REGION Network 2: Manual Operation Cm - typeAxis64PosInterface
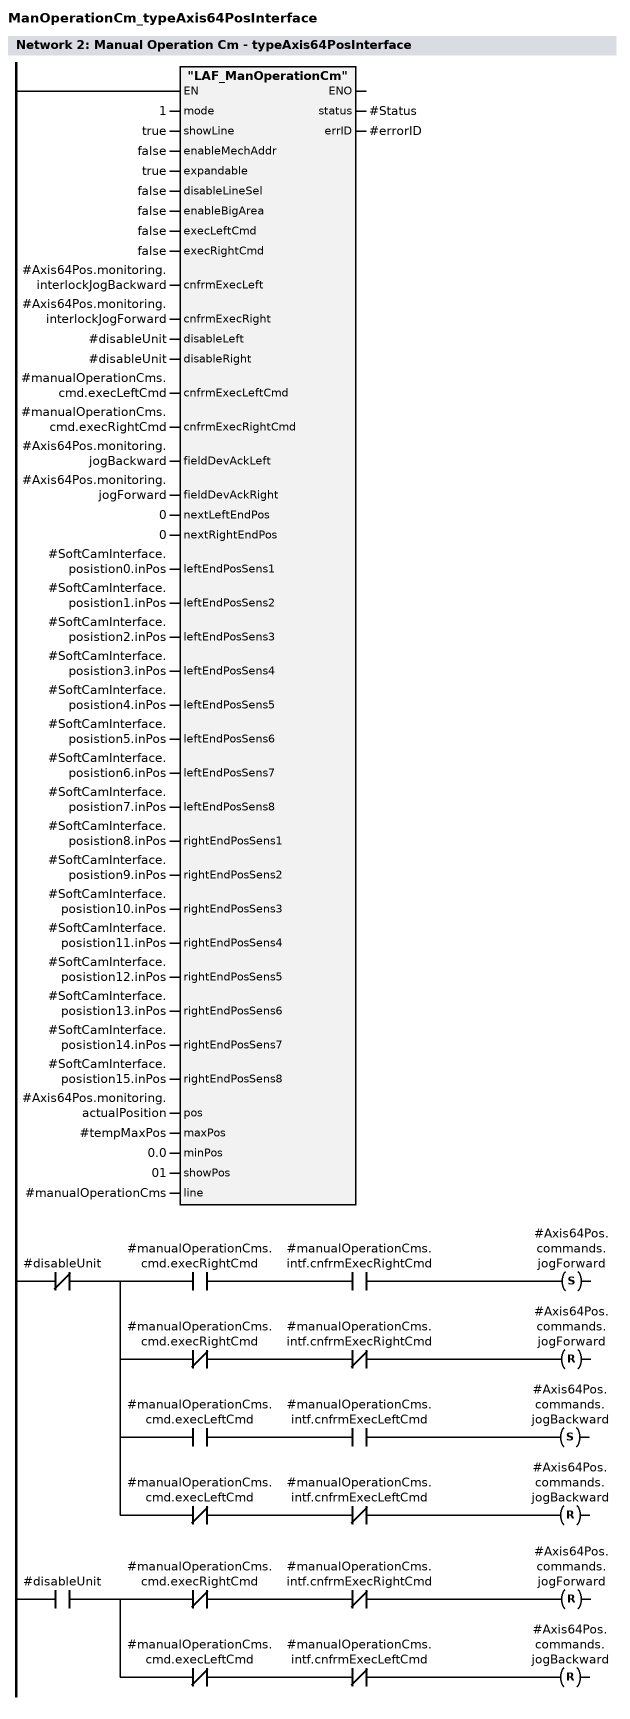
   RUNG wire#powerrail
      "LAF_ManOperationCm"(mode := 1, showLine := true, enableMechAddr := false, expandable := true, disableLineSel := false, enableBigArea := false, execLeftCmd := false, execRightCmd := false, cnfrmExecLeft := #Axis64Pos.monitoring.interlockJogBackward, cnfrmExecRight := #Axis64Pos.monitoring.interlockJogForward, disableLeft := #disableUnit, disableRight := #disableUnit, cnfrmExecLeftCmd := #manualOperationCms.cmd.execLeftCmd, cnfrmExecRightCmd := #manualOperationCms.cmd.execRightCmd, fieldDevAckLeft := #Axis64Pos.monitoring.jogBackward, fieldDevAckRight := #Axis64Pos.monitoring.jogForward, nextLeftEndPos := 0, nextRightEndPos := 0, leftEndPosSens1 := #SoftCamInterface.posistion0.inPos, leftEndPosSens2 := #SoftCamInterface.posistion1.inPos, leftEndPosSens3 := #SoftCamInterface.posistion2.inPos, leftEndPosSens4 := #SoftCamInterface.posistion3.inPos, leftEndPosSens5 := #SoftCamInterface.posistion4.inPos, leftEndPosSens6 := #SoftCamInterface.posistion5.inPos, leftEndPosSens7 := #SoftCamInterface.posistion6.inPos, leftEndPosSens8 := #SoftCamInterface.posistion7.inPos, rightEndPosSens1 := #SoftCamInterface.posistion8.inPos, rightEndPosSens2 := #SoftCamInterface.posistion9.inPos, rightEndPosSens3 := #SoftCamInterface.posistion10.inPos, rightEndPosSens4 := #SoftCamInterface.posistion11.inPos, rightEndPosSens5 := #SoftCamInterface.posistion12.inPos, rightEndPosSens6 := #SoftCamInterface.posistion13.inPos, rightEndPosSens7 := #SoftCamInterface.posistion14.inPos, rightEndPosSens8 := #SoftCamInterface.posistion15.inPos, pos := #Axis64Pos.monitoring.actualPosition, maxPos := #tempMaxPos, minPos := 0.0, showPos := 01, line := #manualOperationCms, status => #Status, errID => #errorID)
   END_RUNG
   RUNG wire#powerrail
      I_Contact( #disableUnit )
      wire#w1
      Contact( #manualOperationCms.cmd.execRightCmd )
      Contact( #manualOperationCms.intf.cnfrmExecRightCmd )
      S_Coil( #Axis64Pos.commands.jogForward )
   END_RUNG
   RUNG wire#w1
      I_Contact( #manualOperationCms.cmd.execRightCmd )
      I_Contact( #manualOperationCms.intf.cnfrmExecRightCmd )
      R_Coil( #Axis64Pos.commands.jogForward )
   END_RUNG
   RUNG wire#w1
      Contact( #manualOperationCms.cmd.execLeftCmd )
      Contact( #manualOperationCms.intf.cnfrmExecLeftCmd )
      S_Coil( #Axis64Pos.commands.jogBackward )
   END_RUNG
   RUNG wire#w1
      I_Contact( #manualOperationCms.cmd.execLeftCmd )
      I_Contact( #manualOperationCms.intf.cnfrmExecLeftCmd )
      R_Coil( #Axis64Pos.commands.jogBackward )
   END_RUNG
   RUNG wire#powerrail
      Contact( #disableUnit )
      wire#w2
      I_Contact( #manualOperationCms.cmd.execRightCmd )
      I_Contact( #manualOperationCms.intf.cnfrmExecRightCmd )
      R_Coil( #Axis64Pos.commands.jogForward )
   END_RUNG
   RUNG wire#w2
      I_Contact( #manualOperationCms.cmd.execLeftCmd )
      I_Contact( #manualOperationCms.intf.cnfrmExecLeftCmd )
      R_Coil( #Axis64Pos.commands.jogBackward )
   END_RUNG
   // the same network as SCL:
   "LAF_ManOperationCm"(mode := 1,
                        showLine := true,
                        enableMechAddr := false,
                        expandable := true,
                        disableLineSel := false,
                        enableBigArea := false,
                        execLeftCmd := false,
                        execRightCmd := false,
                        cnfrmExecLeft := #Axis64Pos.monitoring.interlockJogBackward,
                        cnfrmExecRight := #Axis64Pos.monitoring.interlockJogForward,
                        disableLeft := #disableUnit,
                        disableRight := #disableUnit,
                        cnfrmExecLeftCmd := #manualOperationCms.cmd.execLeftCmd,
                        cnfrmExecRightCmd := #manualOperationCms.cmd.execRightCmd,
                        fieldDevAckLeft := #Axis64Pos.monitoring.jogBackward,
                        fieldDevAckRight := #Axis64Pos.monitoring.jogForward,
                        nextLeftEndPos := 0,
                        nextRightEndPos := 0,
                        leftEndPosSens1 := #SoftCamInterface.posistion0.inPos,
                        leftEndPosSens2 := #SoftCamInterface.posistion1.inPos,
                        leftEndPosSens3 := #SoftCamInterface.posistion2.inPos,
                        leftEndPosSens4 := #SoftCamInterface.posistion3.inPos,
                        leftEndPosSens5 := #SoftCamInterface.posistion4.inPos,
                        leftEndPosSens6 := #SoftCamInterface.posistion5.inPos,
                        leftEndPosSens7 := #SoftCamInterface.posistion6.inPos,
                        leftEndPosSens8 := #SoftCamInterface.posistion7.inPos,
                        rightEndPosSens1 := #SoftCamInterface.posistion8.inPos,
                        rightEndPosSens2 := #SoftCamInterface.posistion9.inPos,
                        rightEndPosSens3 := #SoftCamInterface.posistion10.inPos,
                        rightEndPosSens4 := #SoftCamInterface.posistion11.inPos,
                        rightEndPosSens5 := #SoftCamInterface.posistion12.inPos,
                        rightEndPosSens6 := #SoftCamInterface.posistion13.inPos,
                        rightEndPosSens7 := #SoftCamInterface.posistion14.inPos,
                        rightEndPosSens8 := #SoftCamInterface.posistion15.inPos,
                        pos := #Axis64Pos.monitoring.actualPosition,
                        maxPos := #tempMaxPos,
                        minPos := 0.0,
                        showPos := 01,
                        line := #manualOperationCms,
                        status => #Status,
                        errID => #errorID);
   IF NOT #disableUnit AND #manualOperationCms.cmd.execRightCmd AND #manualOperationCms.intf.cnfrmExecRightCmd THEN
       #Axis64Pos.commands.jogForward := TRUE;
   END_IF;
   IF NOT #disableUnit AND NOT #manualOperationCms.cmd.execRightCmd AND NOT #manualOperationCms.intf.cnfrmExecRightCmd THEN
       #Axis64Pos.commands.jogForward := FALSE;
   END_IF;
   IF NOT #disableUnit AND #manualOperationCms.cmd.execLeftCmd AND #manualOperationCms.intf.cnfrmExecLeftCmd THEN
       #Axis64Pos.commands.jogBackward := TRUE;
   END_IF;
   IF NOT #disableUnit AND NOT #manualOperationCms.cmd.execLeftCmd AND NOT #manualOperationCms.intf.cnfrmExecLeftCmd THEN
       #Axis64Pos.commands.jogBackward := FALSE;
   END_IF;
   IF #disableUnit AND NOT #manualOperationCms.cmd.execRightCmd AND NOT #manualOperationCms.intf.cnfrmExecRightCmd THEN
       #Axis64Pos.commands.jogForward := FALSE;
   END_IF;
   IF #disableUnit AND NOT #manualOperationCms.cmd.execLeftCmd AND NOT #manualOperationCms.intf.cnfrmExecLeftCmd THEN
       #Axis64Pos.commands.jogBackward := FALSE;
   END_IF;
END_REGION
END_FUNCTION

FUNCTION "ManOperationCm_typeTwoWayActuatorInterface" : Void   // FC65, LAD
// stored: SetENOAutomatically false
   VAR_INPUT
      disableUnit : Bool;
   END_VAR
   VAR_OUTPUT
      Status : Word;
      errorID : Word;
   END_VAR
   VAR_IN_OUT
      manualOperationEm : "LAF_typeManEm";
      manualOperationEmArea : "LAF_typeManOperationArea";
      manualOperationCms : "LAF_typeManOperation";
      twoWayAcutor : "LBC_typeTwoWayActuatorInterface";
   END_VAR
BEGIN

REGION Network 1: Manual Operation Cm - typeTwoWayActuatorInterface
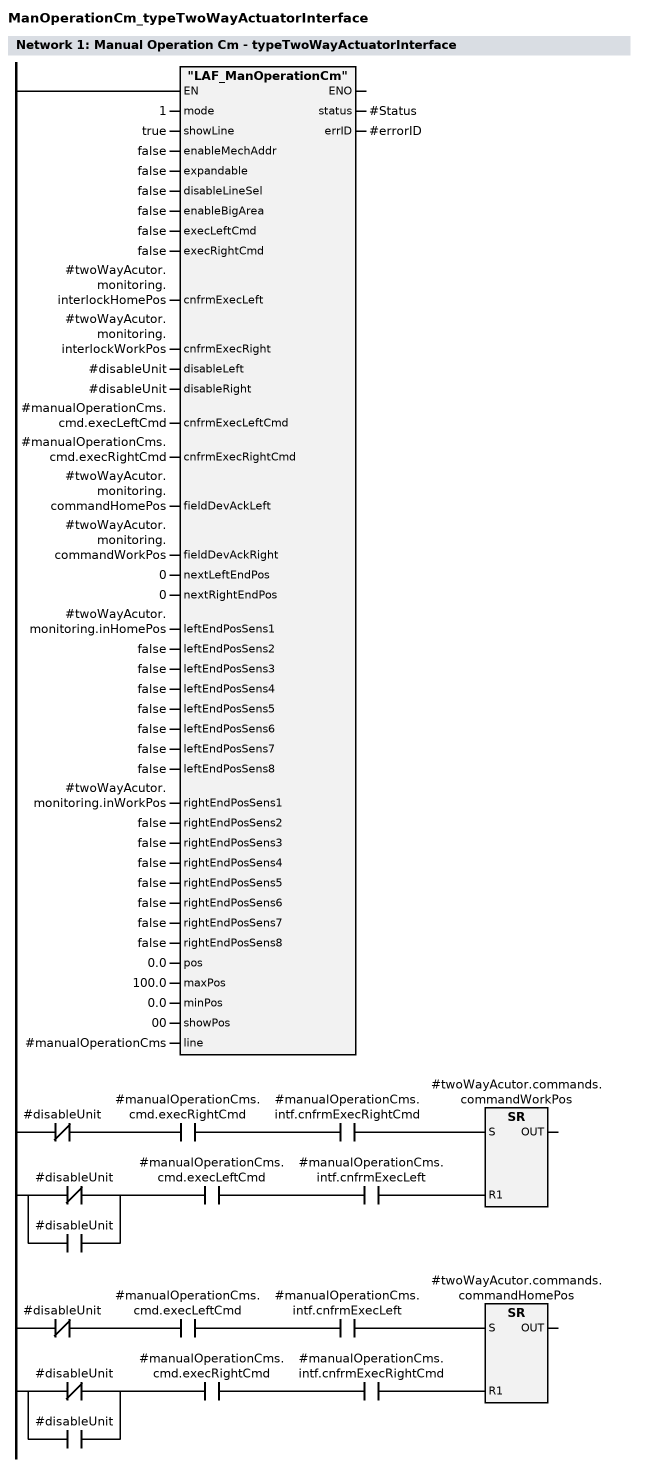
   RUNG wire#powerrail
      "LAF_ManOperationCm"(mode := 1, showLine := true, enableMechAddr := false, expandable := false, disableLineSel := false, enableBigArea := false, execLeftCmd := false, execRightCmd := false, cnfrmExecLeft := #twoWayAcutor.monitoring.interlockHomePos, cnfrmExecRight := #twoWayAcutor.monitoring.interlockWorkPos, disableLeft := #disableUnit, disableRight := #disableUnit, cnfrmExecLeftCmd := #manualOperationCms.cmd.execLeftCmd, cnfrmExecRightCmd := #manualOperationCms.cmd.execRightCmd, fieldDevAckLeft := #twoWayAcutor.monitoring.commandHomePos, fieldDevAckRight := #twoWayAcutor.monitoring.commandWorkPos, nextLeftEndPos := 0, nextRightEndPos := 0, leftEndPosSens1 := #twoWayAcutor.monitoring.inHomePos, leftEndPosSens2 := false, leftEndPosSens3 := false, leftEndPosSens4 := false, leftEndPosSens5 := false, leftEndPosSens6 := false, leftEndPosSens7 := false, leftEndPosSens8 := false, rightEndPosSens1 := #twoWayAcutor.monitoring.inWorkPos, rightEndPosSens2 := false, rightEndPosSens3 := false, rightEndPosSens4 := false, rightEndPosSens5 := false, rightEndPosSens6 := false, rightEndPosSens7 := false, rightEndPosSens8 := false, pos := 0.0, maxPos := 100.0, minPos := 0.0, showPos := 00, line := #manualOperationCms, status => #Status, errID => #errorID)
   END_RUNG
   RUNG wire#powerrail
      I_Contact( #disableUnit )
      Contact( #manualOperationCms.cmd.execRightCmd )
      Contact( #manualOperationCms.intf.cnfrmExecRightCmd )
      S_SR(operand := #twoWayAcutor.commands.commandWorkPos, r1 := wire#w2)
   END_RUNG
   RUNG wire#powerrail
      I_Contact( #disableUnit )
      wire#w1
      Contact( #manualOperationCms.cmd.execLeftCmd )
      Contact( #manualOperationCms.intf.cnfrmExecLeft )
   END_RUNG wire#w2
   RUNG wire#powerrail
      Contact( #disableUnit )
   END_RUNG wire#w1
   RUNG wire#powerrail
      I_Contact( #disableUnit )
      Contact( #manualOperationCms.cmd.execLeftCmd )
      Contact( #manualOperationCms.intf.cnfrmExecLeft )
      S_SR(operand := #twoWayAcutor.commands.commandHomePos, r1 := wire#w4)
   END_RUNG
   RUNG wire#powerrail
      I_Contact( #disableUnit )
      wire#w3
      Contact( #manualOperationCms.cmd.execRightCmd )
      Contact( #manualOperationCms.intf.cnfrmExecRightCmd )
   END_RUNG wire#w4
   RUNG wire#powerrail
      Contact( #disableUnit )
   END_RUNG wire#w3
   // the same network as SCL:
   "LAF_ManOperationCm"(mode := 1,
                        showLine := true,
                        enableMechAddr := false,
                        expandable := false,
                        disableLineSel := false,
                        enableBigArea := false,
                        execLeftCmd := false,
                        execRightCmd := false,
                        cnfrmExecLeft := #twoWayAcutor.monitoring.interlockHomePos,
                        cnfrmExecRight := #twoWayAcutor.monitoring.interlockWorkPos,
                        disableLeft := #disableUnit,
                        disableRight := #disableUnit,
                        cnfrmExecLeftCmd := #manualOperationCms.cmd.execLeftCmd,
                        cnfrmExecRightCmd := #manualOperationCms.cmd.execRightCmd,
                        fieldDevAckLeft := #twoWayAcutor.monitoring.commandHomePos,
                        fieldDevAckRight := #twoWayAcutor.monitoring.commandWorkPos,
                        nextLeftEndPos := 0,
                        nextRightEndPos := 0,
                        leftEndPosSens1 := #twoWayAcutor.monitoring.inHomePos,
                        leftEndPosSens2 := false,
                        leftEndPosSens3 := false,
                        leftEndPosSens4 := false,
                        leftEndPosSens5 := false,
                        leftEndPosSens6 := false,
                        leftEndPosSens7 := false,
                        leftEndPosSens8 := false,
                        rightEndPosSens1 := #twoWayAcutor.monitoring.inWorkPos,
                        rightEndPosSens2 := false,
                        rightEndPosSens3 := false,
                        rightEndPosSens4 := false,
                        rightEndPosSens5 := false,
                        rightEndPosSens6 := false,
                        rightEndPosSens7 := false,
                        rightEndPosSens8 := false,
                        pos := 0.0,
                        maxPos := 100.0,
                        minPos := 0.0,
                        showPos := 00,
                        line := #manualOperationCms,
                        status => #Status,
                        errID => #errorID);
   IF NOT #disableUnit AND #manualOperationCms.cmd.execRightCmd AND #manualOperationCms.intf.cnfrmExecRightCmd THEN
       #twoWayAcutor.commands.commandWorkPos := TRUE;   // SR flip-flop
   END_IF;
   IF (NOT #disableUnit OR #disableUnit) AND #manualOperationCms.cmd.execLeftCmd AND #manualOperationCms.intf.cnfrmExecLeft THEN
       #twoWayAcutor.commands.commandWorkPos := FALSE;
   END_IF;
   IF NOT #disableUnit AND #manualOperationCms.cmd.execLeftCmd AND #manualOperationCms.intf.cnfrmExecLeft THEN
       #twoWayAcutor.commands.commandHomePos := TRUE;   // SR flip-flop
   END_IF;
   IF (NOT #disableUnit OR #disableUnit) AND #manualOperationCms.cmd.execRightCmd AND #manualOperationCms.intf.cnfrmExecRightCmd THEN
       #twoWayAcutor.commands.commandHomePos := FALSE;
   END_IF;
END_REGION
END_FUNCTION

FUNCTION "CallDiagnostic" : Void   // FC16, LAD
TITLE = Diagnostics
AUTHOR : SICAR
FAMILY : Diag
// Call of SICAR Diagnostic blocks
// stored: IsIECCheckEnabled true, SetENOAutomatically true
   VAR_TEMP
      statWStringName : WString[24];
      tempHardwareOKexample : Bool;   // REPLACE: This output can be used as an interlock for Control Modules
   END_VAR
   VAR CONSTANT
      TRUE : Bool := TRUE;
   END_VAR
   // Ret_Val : Ret_Val
   VAR_TEMP   // added for the SCL form of the ladder/FBD networks
      _w1 : Bool;
   END_VAR
BEGIN

REGION Network 1: BLOCK INFO HEADER
   // SIEMENS AG / (c)Copyright 2023
   // ------------------------------------------------------------------------------
   // Title:            CallDiagnostic (FC16)
   // Comment/Function: Call of SICAR Diagnostic blocks
   // Library/Family:   Diag
   // Author:           SICAR
   // Tested with:      ---
   // Engineering:      TIA Portal V19
   // Restrictions:     -
   // Requirements:     ---
   // ------------------------------------------------------------------------------
   // Change log table:
   // Version | Date | Expert in charge | Changes applied
   // -------|---------|-------------|--------------------------------------------
   // 01.00.00 | 01.01.1999 | Person x | First released version
   // 01.00.01 | 02.01.1999 | Person y | Block was Updated
END_REGION

REGION Network 2: Call: Diagnostic Profinet Devices
   // For diagnose the whole profinet devices of this PLC
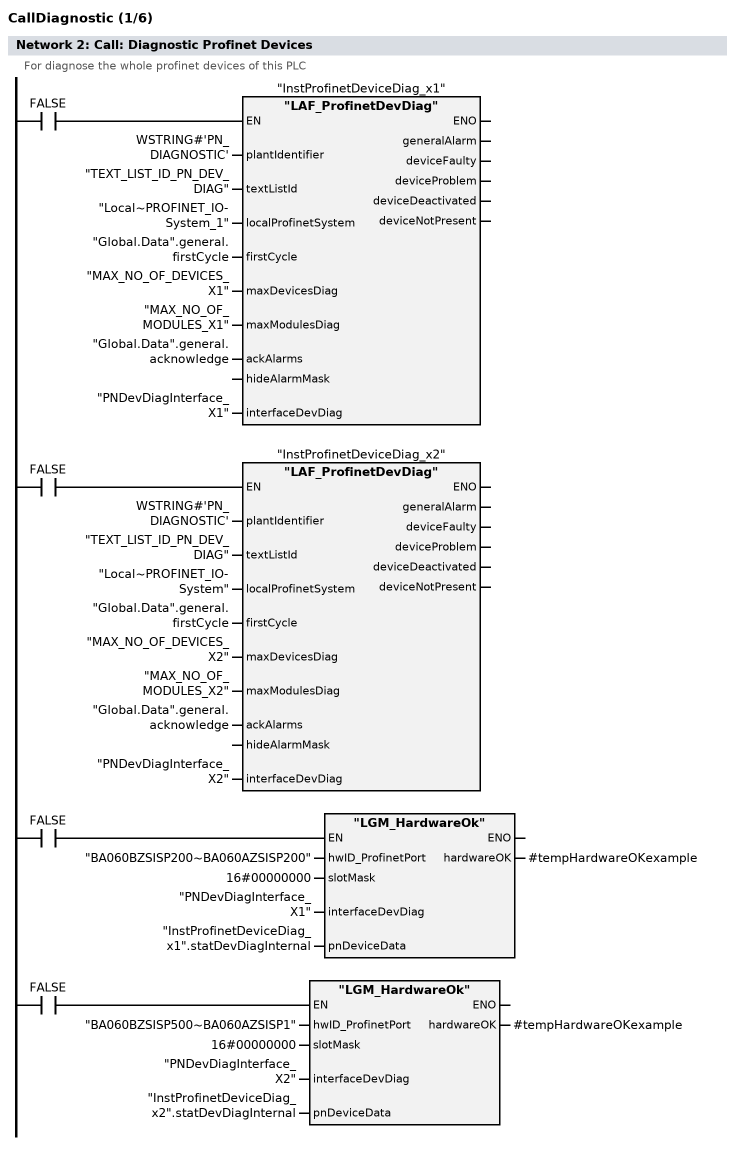
   RUNG wire#powerrail
      Contact( FALSE )
      "InstProfinetDeviceDiag_x1"(plantIdentifier := WSTRING#'PN_DIAGNOSTIC', textListId := "TEXT_LIST_ID_PN_DEV_DIAG", localProfinetSystem := "Local~PROFINET_IO-System_1", firstCycle := "Global.Data".general.firstCycle, maxDevicesDiag := "MAX_NO_OF_DEVICES_X1", maxModulesDiag := "MAX_NO_OF_MODULES_X1", ackAlarms := "Global.Data".general.acknowledge, hideAlarmMask :=, interfaceDevDiag := "PNDevDiagInterface_X1", generalAlarm =>, deviceFaulty =>, deviceProblem =>, deviceDeactivated =>, deviceNotPresent =>)
   END_RUNG
   RUNG wire#powerrail
      Contact( FALSE )
      "InstProfinetDeviceDiag_x2"(plantIdentifier := WSTRING#'PN_DIAGNOSTIC', textListId := "TEXT_LIST_ID_PN_DEV_DIAG", localProfinetSystem := "Local~PROFINET_IO-System", firstCycle := "Global.Data".general.firstCycle, maxDevicesDiag := "MAX_NO_OF_DEVICES_X2", maxModulesDiag := "MAX_NO_OF_MODULES_X2", ackAlarms := "Global.Data".general.acknowledge, hideAlarmMask :=, interfaceDevDiag := "PNDevDiagInterface_X2", generalAlarm =>, deviceFaulty =>, deviceProblem =>, deviceDeactivated =>, deviceNotPresent =>)
   END_RUNG
   RUNG wire#powerrail
      Contact( FALSE )
      "LGM_HardwareOk"(hwID_ProfinetPort := "BA060BZSISP200~BA060AZSISP200", slotMask := 16#00000000, interfaceDevDiag := "PNDevDiagInterface_X1", pnDeviceData := "InstProfinetDeviceDiag_x1".statDevDiagInternal, hardwareOK => #tempHardwareOKexample)
   END_RUNG
   RUNG wire#powerrail
      Contact( FALSE )
      "LGM_HardwareOk"(hwID_ProfinetPort := "BA060BZSISP500~BA060AZSISP1", slotMask := 16#00000000, interfaceDevDiag := "PNDevDiagInterface_X2", pnDeviceData := "InstProfinetDeviceDiag_x2".statDevDiagInternal, hardwareOK => #tempHardwareOKexample)
   END_RUNG
   // the same network as SCL:
   IF FALSE THEN
       "InstProfinetDeviceDiag_x1"(plantIdentifier := WSTRING#'PN_DIAGNOSTIC',   // "LAF_ProfinetDevDiag"
                               textListId := "TEXT_LIST_ID_PN_DEV_DIAG",
                               localProfinetSystem := "Local~PROFINET_IO-System_1",
                               firstCycle := "Global.Data".general.firstCycle,
                               maxDevicesDiag := "MAX_NO_OF_DEVICES_X1",
                               maxModulesDiag := "MAX_NO_OF_MODULES_X1",
                               ackAlarms := "Global.Data".general.acknowledge,
                               interfaceDevDiag := "PNDevDiagInterface_X1");
       "InstProfinetDeviceDiag_x2"(plantIdentifier := WSTRING#'PN_DIAGNOSTIC',   // "LAF_ProfinetDevDiag"
                               textListId := "TEXT_LIST_ID_PN_DEV_DIAG",
                               localProfinetSystem := "Local~PROFINET_IO-System",
                               firstCycle := "Global.Data".general.firstCycle,
                               maxDevicesDiag := "MAX_NO_OF_DEVICES_X2",
                               maxModulesDiag := "MAX_NO_OF_MODULES_X2",
                               ackAlarms := "Global.Data".general.acknowledge,
                               interfaceDevDiag := "PNDevDiagInterface_X2");
       "LGM_HardwareOk"(hwID_ProfinetPort := "BA060BZSISP200~BA060AZSISP200",
                        slotMask := 16#00000000,
                        interfaceDevDiag := "PNDevDiagInterface_X1",
                        pnDeviceData := "InstProfinetDeviceDiag_x1".statDevDiagInternal,
                        hardwareOK => #tempHardwareOKexample);
       "LGM_HardwareOk"(hwID_ProfinetPort := "BA060BZSISP500~BA060AZSISP1",
                        slotMask := 16#00000000,
                        interfaceDevDiag := "PNDevDiagInterface_X2",
                        pnDeviceData := "InstProfinetDeviceDiag_x2".statDevDiagInternal,
                        hardwareOK => #tempHardwareOKexample);
   END_IF;
END_REGION

REGION Network 3: Call: Diagnostic Bool Interface Signals
   // Call the interface bool blocks to show boolean signals on the HMI
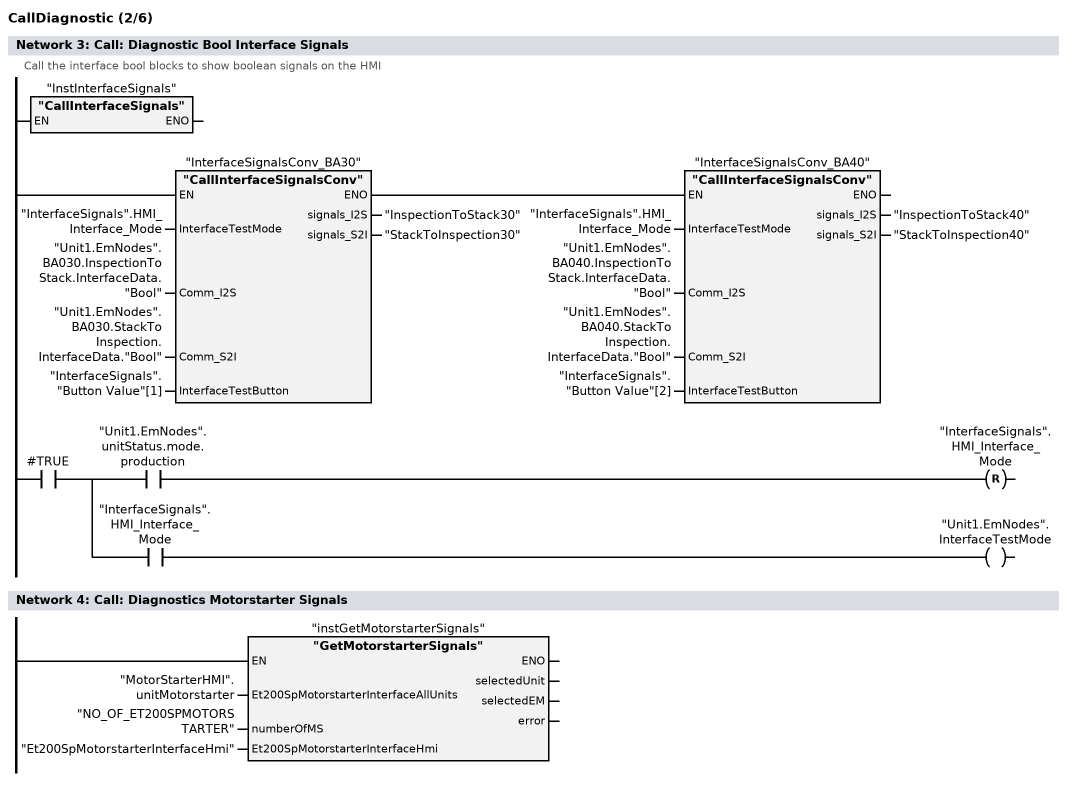
   RUNG wire#powerrail
      "InstInterfaceSignals"()
   END_RUNG
   RUNG wire#powerrail
      "InterfaceSignalsConv_BA30"(InterfaceTestMode := "InterfaceSignals".HMI_Interface_Mode, Comm_I2S := "Unit1.EmNodes".BA030.InspectionToStack.InterfaceData."Bool", Comm_S2I := "Unit1.EmNodes".BA030.StackToInspection.InterfaceData."Bool", InterfaceTestButton := "InterfaceSignals"."Button Value"[1], signals_I2S => "InspectionToStack30", signals_S2I => "StackToInspection30")
      "InterfaceSignalsConv_BA40"(InterfaceTestMode := "InterfaceSignals".HMI_Interface_Mode, Comm_I2S := "Unit1.EmNodes".BA040.InspectionToStack.InterfaceData."Bool", Comm_S2I := "Unit1.EmNodes".BA040.StackToInspection.InterfaceData."Bool", InterfaceTestButton := "InterfaceSignals"."Button Value"[2], signals_I2S => "InspectionToStack40", signals_S2I => "StackToInspection40")
   END_RUNG
   RUNG wire#powerrail
      Contact( #TRUE )
      wire#w1
      Contact( "Unit1.EmNodes".unitStatus.mode.production )
      R_Coil( "InterfaceSignals".HMI_Interface_Mode )
   END_RUNG
   RUNG wire#w1
      Contact( "InterfaceSignals".HMI_Interface_Mode )
      Coil( "Unit1.EmNodes".InterfaceTestMode )
   END_RUNG
   // the same network as SCL:
   "InstInterfaceSignals"();   // "CallInterfaceSignals"
   "InterfaceSignalsConv_BA30"(InterfaceTestMode := "InterfaceSignals".HMI_Interface_Mode,   // "CallInterfaceSignalsConv"
                           Comm_I2S := "Unit1.EmNodes".BA030.InspectionToStack.InterfaceData."Bool",
                           Comm_S2I := "Unit1.EmNodes".BA030.StackToInspection.InterfaceData."Bool",
                           InterfaceTestButton := "InterfaceSignals"."Button Value"[1],
                           signals_I2S => "InspectionToStack30",
                           signals_S2I => "StackToInspection30",
                           ENO => #_w1);
   IF #_w1 THEN
       "InterfaceSignalsConv_BA40"(InterfaceTestMode := "InterfaceSignals".HMI_Interface_Mode,   // "CallInterfaceSignalsConv"
                               Comm_I2S := "Unit1.EmNodes".BA040.InspectionToStack.InterfaceData."Bool",
                               Comm_S2I := "Unit1.EmNodes".BA040.StackToInspection.InterfaceData."Bool",
                               InterfaceTestButton := "InterfaceSignals"."Button Value"[2],
                               signals_I2S => "InspectionToStack40",
                               signals_S2I => "StackToInspection40");
   END_IF;
   IF #TRUE AND "Unit1.EmNodes".unitStatus.mode.production THEN
       "InterfaceSignals".HMI_Interface_Mode := FALSE;
   END_IF;
   "Unit1.EmNodes".InterfaceTestMode := #TRUE AND "InterfaceSignals".HMI_Interface_Mode;
END_REGION

REGION Network 4: Call: Diagnostics Motorstarter Signals
   RUNG wire#powerrail
      "instGetMotorstarterSignals"(Et200SpMotorstarterInterfaceAllUnits := "MotorStarterHMI".unitMotorstarter, numberOfMS := "NO_OF_ET200SPMOTORSTARTER", Et200SpMotorstarterInterfaceHmi := "Et200SpMotorstarterInterfaceHmi", selectedUnit =>, selectedEM =>, error =>)
   END_RUNG
   // the same network as SCL:
   "instGetMotorstarterSignals"(Et200SpMotorstarterInterfaceAllUnits := "MotorStarterHMI".unitMotorstarter,   // "GetMotorstarterSignals"
                           numberOfMS := "NO_OF_ET200SPMOTORSTARTER",
                           Et200SpMotorstarterInterfaceHmi := "Et200SpMotorstarterInterfaceHmi");
END_REGION

REGION Network 5: Call: Diagnostics Drives
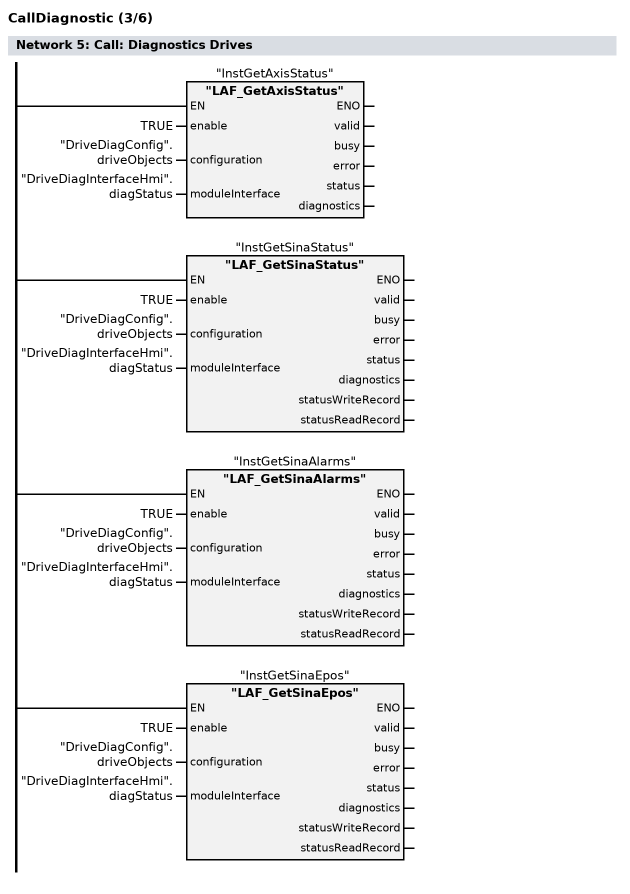
   RUNG wire#powerrail
      "InstGetAxisStatus"(enable := TRUE, configuration := "DriveDiagConfig".driveObjects, moduleInterface := "DriveDiagInterfaceHmi".diagStatus, valid =>, busy =>, error =>, status =>, diagnostics =>)
   END_RUNG
   RUNG wire#powerrail
      "InstGetSinaStatus"(enable := TRUE, configuration := "DriveDiagConfig".driveObjects, moduleInterface := "DriveDiagInterfaceHmi".diagStatus, valid =>, busy =>, error =>, status =>, diagnostics =>, statusWriteRecord =>, statusReadRecord =>)
   END_RUNG
   RUNG wire#powerrail
      "InstGetSinaAlarms"(enable := TRUE, configuration := "DriveDiagConfig".driveObjects, moduleInterface := "DriveDiagInterfaceHmi".diagStatus, valid =>, busy =>, error =>, status =>, diagnostics =>, statusWriteRecord =>, statusReadRecord =>)
   END_RUNG
   RUNG wire#powerrail
      "InstGetSinaEpos"(enable := TRUE, configuration := "DriveDiagConfig".driveObjects, moduleInterface := "DriveDiagInterfaceHmi".diagStatus, valid =>, busy =>, error =>, status =>, diagnostics =>, statusWriteRecord =>, statusReadRecord =>)
   END_RUNG
   // the same network as SCL:
   "InstGetAxisStatus"(enable := TRUE,   // "LAF_GetAxisStatus"
                       configuration := "DriveDiagConfig".driveObjects,
                       moduleInterface := "DriveDiagInterfaceHmi".diagStatus);
   "InstGetSinaStatus"(enable := TRUE,   // "LAF_GetSinaStatus"
                       configuration := "DriveDiagConfig".driveObjects,
                       moduleInterface := "DriveDiagInterfaceHmi".diagStatus);
   "InstGetSinaAlarms"(enable := TRUE,   // "LAF_GetSinaAlarms"
                       configuration := "DriveDiagConfig".driveObjects,
                       moduleInterface := "DriveDiagInterfaceHmi".diagStatus);
   "InstGetSinaEpos"(enable := TRUE,   // "LAF_GetSinaEpos"
                     configuration := "DriveDiagConfig".driveObjects,
                     moduleInterface := "DriveDiagInterfaceHmi".diagStatus);
END_REGION

REGION Network 6: Call: Servo Torque Cal (DR1~10)
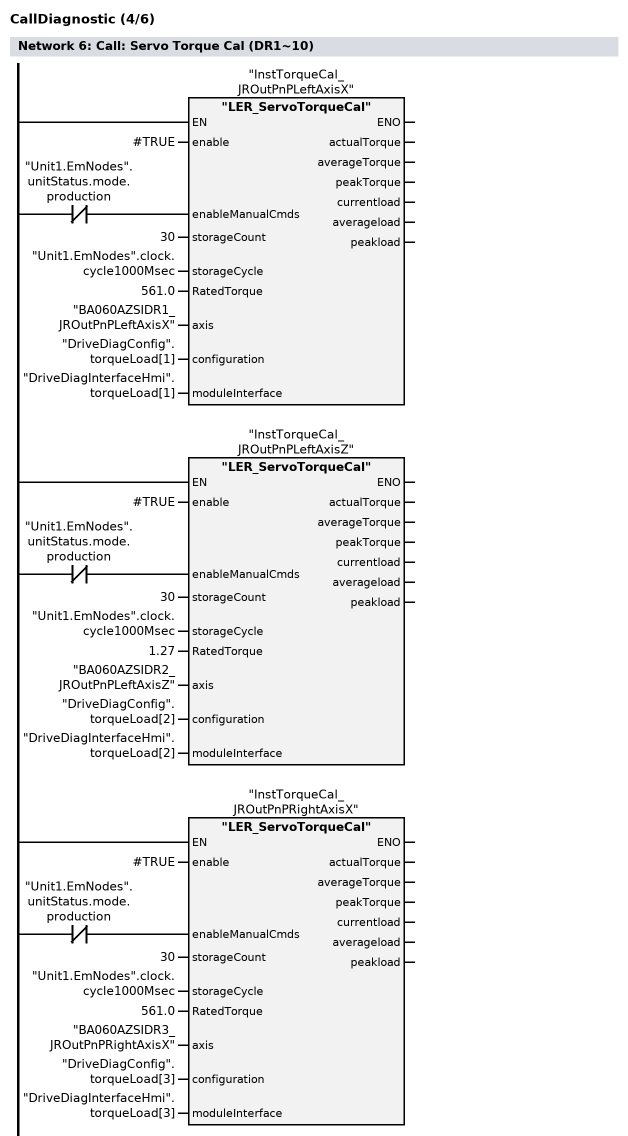
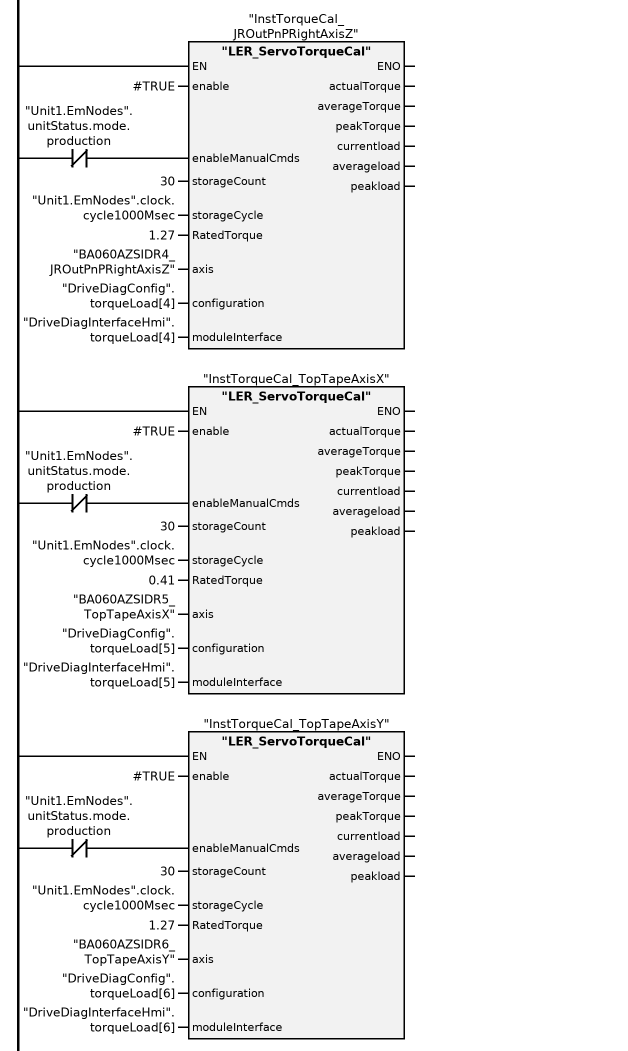
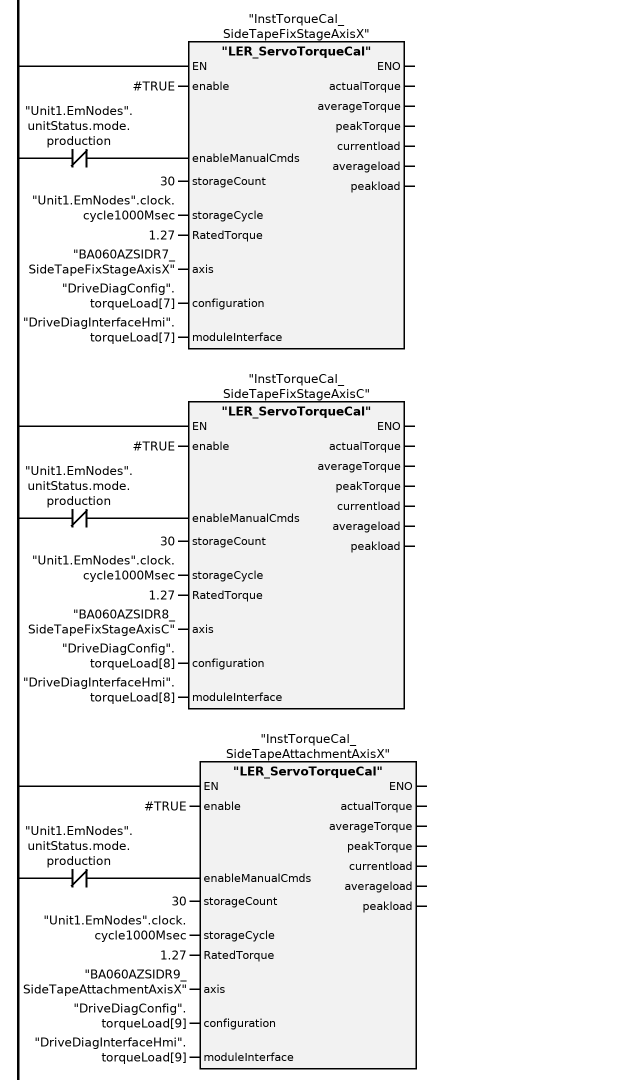
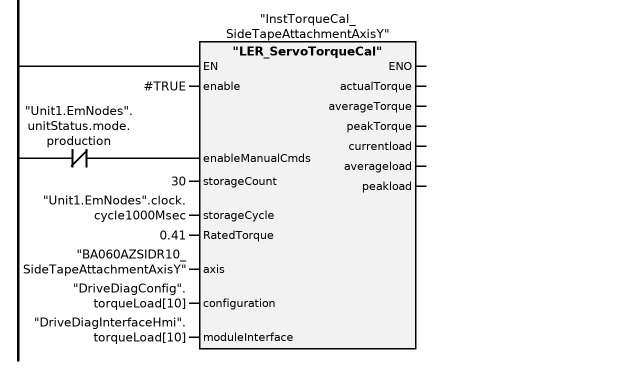
   RUNG wire#powerrail
      "InstTorqueCal_JROutPnPLeftAxisX"(enableManualCmds := wire#w1, enable := #TRUE, storageCount := 30, storageCycle := "Unit1.EmNodes".clock.cycle1000Msec, RatedTorque := 561.0, axis := "BA060AZSIDR1_JROutPnPLeftAxisX", configuration := "DriveDiagConfig".torqueLoad[1], moduleInterface := "DriveDiagInterfaceHmi".torqueLoad[1], actualTorque =>, averageTorque =>, peakTorque =>, currentload =>, averageload =>, peakload =>)
   END_RUNG
   RUNG wire#powerrail
      I_Contact( "Unit1.EmNodes".unitStatus.mode.production )
   END_RUNG wire#w1
   RUNG wire#powerrail
      "InstTorqueCal_JROutPnPLeftAxisZ"(enableManualCmds := wire#w2, enable := #TRUE, storageCount := 30, storageCycle := "Unit1.EmNodes".clock.cycle1000Msec, RatedTorque := 1.27, axis := "BA060AZSIDR2_JROutPnPLeftAxisZ", configuration := "DriveDiagConfig".torqueLoad[2], moduleInterface := "DriveDiagInterfaceHmi".torqueLoad[2], actualTorque =>, averageTorque =>, peakTorque =>, currentload =>, averageload =>, peakload =>)
   END_RUNG
   RUNG wire#powerrail
      I_Contact( "Unit1.EmNodes".unitStatus.mode.production )
   END_RUNG wire#w2
   RUNG wire#powerrail
      "InstTorqueCal_JROutPnPRightAxisX"(enableManualCmds := wire#w3, enable := #TRUE, storageCount := 30, storageCycle := "Unit1.EmNodes".clock.cycle1000Msec, RatedTorque := 561.0, axis := "BA060AZSIDR3_JROutPnPRightAxisX", configuration := "DriveDiagConfig".torqueLoad[3], moduleInterface := "DriveDiagInterfaceHmi".torqueLoad[3], actualTorque =>, averageTorque =>, peakTorque =>, currentload =>, averageload =>, peakload =>)
   END_RUNG
   RUNG wire#powerrail
      I_Contact( "Unit1.EmNodes".unitStatus.mode.production )
   END_RUNG wire#w3
   RUNG wire#powerrail
      "InstTorqueCal_JROutPnPRightAxisZ"(enableManualCmds := wire#w4, enable := #TRUE, storageCount := 30, storageCycle := "Unit1.EmNodes".clock.cycle1000Msec, RatedTorque := 1.27, axis := "BA060AZSIDR4_JROutPnPRightAxisZ", configuration := "DriveDiagConfig".torqueLoad[4], moduleInterface := "DriveDiagInterfaceHmi".torqueLoad[4], actualTorque =>, averageTorque =>, peakTorque =>, currentload =>, averageload =>, peakload =>)
   END_RUNG
   RUNG wire#powerrail
      I_Contact( "Unit1.EmNodes".unitStatus.mode.production )
   END_RUNG wire#w4
   RUNG wire#powerrail
      "InstTorqueCal_TopTapeAxisX"(enableManualCmds := wire#w5, enable := #TRUE, storageCount := 30, storageCycle := "Unit1.EmNodes".clock.cycle1000Msec, RatedTorque := 0.41, axis := "BA060AZSIDR5_TopTapeAxisX", configuration := "DriveDiagConfig".torqueLoad[5], moduleInterface := "DriveDiagInterfaceHmi".torqueLoad[5], actualTorque =>, averageTorque =>, peakTorque =>, currentload =>, averageload =>, peakload =>)
   END_RUNG
   RUNG wire#powerrail
      I_Contact( "Unit1.EmNodes".unitStatus.mode.production )
   END_RUNG wire#w5
   RUNG wire#powerrail
      "InstTorqueCal_TopTapeAxisY"(enableManualCmds := wire#w6, enable := #TRUE, storageCount := 30, storageCycle := "Unit1.EmNodes".clock.cycle1000Msec, RatedTorque := 1.27, axis := "BA060AZSIDR6_TopTapeAxisY", configuration := "DriveDiagConfig".torqueLoad[6], moduleInterface := "DriveDiagInterfaceHmi".torqueLoad[6], actualTorque =>, averageTorque =>, peakTorque =>, currentload =>, averageload =>, peakload =>)
   END_RUNG
   RUNG wire#powerrail
      I_Contact( "Unit1.EmNodes".unitStatus.mode.production )
   END_RUNG wire#w6
   RUNG wire#powerrail
      "InstTorqueCal_SideTapeFixStageAxisX"(enableManualCmds := wire#w7, enable := #TRUE, storageCount := 30, storageCycle := "Unit1.EmNodes".clock.cycle1000Msec, RatedTorque := 1.27, axis := "BA060AZSIDR7_SideTapeFixStageAxisX", configuration := "DriveDiagConfig".torqueLoad[7], moduleInterface := "DriveDiagInterfaceHmi".torqueLoad[7], actualTorque =>, averageTorque =>, peakTorque =>, currentload =>, averageload =>, peakload =>)
   END_RUNG
   RUNG wire#powerrail
      I_Contact( "Unit1.EmNodes".unitStatus.mode.production )
   END_RUNG wire#w7
   RUNG wire#powerrail
      "InstTorqueCal_SideTapeFixStageAxisC"(enableManualCmds := wire#w8, enable := #TRUE, storageCount := 30, storageCycle := "Unit1.EmNodes".clock.cycle1000Msec, RatedTorque := 1.27, axis := "BA060AZSIDR8_SideTapeFixStageAxisC", configuration := "DriveDiagConfig".torqueLoad[8], moduleInterface := "DriveDiagInterfaceHmi".torqueLoad[8], actualTorque =>, averageTorque =>, peakTorque =>, currentload =>, averageload =>, peakload =>)
   END_RUNG
   RUNG wire#powerrail
      I_Contact( "Unit1.EmNodes".unitStatus.mode.production )
   END_RUNG wire#w8
   RUNG wire#powerrail
      "InstTorqueCal_SideTapeAttachmentAxisX"(enableManualCmds := wire#w9, enable := #TRUE, storageCount := 30, storageCycle := "Unit1.EmNodes".clock.cycle1000Msec, RatedTorque := 1.27, axis := "BA060AZSIDR9_SideTapeAttachmentAxisX", configuration := "DriveDiagConfig".torqueLoad[9], moduleInterface := "DriveDiagInterfaceHmi".torqueLoad[9], actualTorque =>, averageTorque =>, peakTorque =>, currentload =>, averageload =>, peakload =>)
   END_RUNG
   RUNG wire#powerrail
      I_Contact( "Unit1.EmNodes".unitStatus.mode.production )
   END_RUNG wire#w9
   RUNG wire#powerrail
      "InstTorqueCal_SideTapeAttachmentAxisY"(enableManualCmds := wire#w10, enable := #TRUE, storageCount := 30, storageCycle := "Unit1.EmNodes".clock.cycle1000Msec, RatedTorque := 0.41, axis := "BA060AZSIDR10_SideTapeAttachmentAxisY", configuration := "DriveDiagConfig".torqueLoad[10], moduleInterface := "DriveDiagInterfaceHmi".torqueLoad[10], actualTorque =>, averageTorque =>, peakTorque =>, currentload =>, averageload =>, peakload =>)
   END_RUNG
   RUNG wire#powerrail
      I_Contact( "Unit1.EmNodes".unitStatus.mode.production )
   END_RUNG wire#w10
   // the same network as SCL:
   "InstTorqueCal_JROutPnPLeftAxisX"(enable := #TRUE,   // "LER_ServoTorqueCal"
                           enableManualCmds := NOT "Unit1.EmNodes".unitStatus.mode.production,
                           storageCount := 30,
                           storageCycle := "Unit1.EmNodes".clock.cycle1000Msec,
                           RatedTorque := 561.0,
                           axis := "BA060AZSIDR1_JROutPnPLeftAxisX",
                           configuration := "DriveDiagConfig".torqueLoad[1],
                           moduleInterface := "DriveDiagInterfaceHmi".torqueLoad[1]);
   "InstTorqueCal_JROutPnPLeftAxisZ"(enable := #TRUE,   // "LER_ServoTorqueCal"
                           enableManualCmds := NOT "Unit1.EmNodes".unitStatus.mode.production,
                           storageCount := 30,
                           storageCycle := "Unit1.EmNodes".clock.cycle1000Msec,
                           RatedTorque := 1.27,
                           axis := "BA060AZSIDR2_JROutPnPLeftAxisZ",
                           configuration := "DriveDiagConfig".torqueLoad[2],
                           moduleInterface := "DriveDiagInterfaceHmi".torqueLoad[2]);
   "InstTorqueCal_JROutPnPRightAxisX"(enable := #TRUE,   // "LER_ServoTorqueCal"
                           enableManualCmds := NOT "Unit1.EmNodes".unitStatus.mode.production,
                           storageCount := 30,
                           storageCycle := "Unit1.EmNodes".clock.cycle1000Msec,
                           RatedTorque := 561.0,
                           axis := "BA060AZSIDR3_JROutPnPRightAxisX",
                           configuration := "DriveDiagConfig".torqueLoad[3],
                           moduleInterface := "DriveDiagInterfaceHmi".torqueLoad[3]);
   "InstTorqueCal_JROutPnPRightAxisZ"(enable := #TRUE,   // "LER_ServoTorqueCal"
                           enableManualCmds := NOT "Unit1.EmNodes".unitStatus.mode.production,
                           storageCount := 30,
                           storageCycle := "Unit1.EmNodes".clock.cycle1000Msec,
                           RatedTorque := 1.27,
                           axis := "BA060AZSIDR4_JROutPnPRightAxisZ",
                           configuration := "DriveDiagConfig".torqueLoad[4],
                           moduleInterface := "DriveDiagInterfaceHmi".torqueLoad[4]);
   "InstTorqueCal_TopTapeAxisX"(enable := #TRUE,   // "LER_ServoTorqueCal"
                           enableManualCmds := NOT "Unit1.EmNodes".unitStatus.mode.production,
                           storageCount := 30,
                           storageCycle := "Unit1.EmNodes".clock.cycle1000Msec,
                           RatedTorque := 0.41,
                           axis := "BA060AZSIDR5_TopTapeAxisX",
                           configuration := "DriveDiagConfig".torqueLoad[5],
                           moduleInterface := "DriveDiagInterfaceHmi".torqueLoad[5]);
   "InstTorqueCal_TopTapeAxisY"(enable := #TRUE,   // "LER_ServoTorqueCal"
                           enableManualCmds := NOT "Unit1.EmNodes".unitStatus.mode.production,
                           storageCount := 30,
                           storageCycle := "Unit1.EmNodes".clock.cycle1000Msec,
                           RatedTorque := 1.27,
                           axis := "BA060AZSIDR6_TopTapeAxisY",
                           configuration := "DriveDiagConfig".torqueLoad[6],
                           moduleInterface := "DriveDiagInterfaceHmi".torqueLoad[6]);
   "InstTorqueCal_SideTapeFixStageAxisX"(enable := #TRUE,   // "LER_ServoTorqueCal"
                           enableManualCmds := NOT "Unit1.EmNodes".unitStatus.mode.production,
                           storageCount := 30,
                           storageCycle := "Unit1.EmNodes".clock.cycle1000Msec,
                           RatedTorque := 1.27,
                           axis := "BA060AZSIDR7_SideTapeFixStageAxisX",
                           configuration := "DriveDiagConfig".torqueLoad[7],
                           moduleInterface := "DriveDiagInterfaceHmi".torqueLoad[7]);
   "InstTorqueCal_SideTapeFixStageAxisC"(enable := #TRUE,   // "LER_ServoTorqueCal"
                           enableManualCmds := NOT "Unit1.EmNodes".unitStatus.mode.production,
                           storageCount := 30,
                           storageCycle := "Unit1.EmNodes".clock.cycle1000Msec,
                           RatedTorque := 1.27,
                           axis := "BA060AZSIDR8_SideTapeFixStageAxisC",
                           configuration := "DriveDiagConfig".torqueLoad[8],
                           moduleInterface := "DriveDiagInterfaceHmi".torqueLoad[8]);
   "InstTorqueCal_SideTapeAttachmentAxisX"(enable := #TRUE,   // "LER_ServoTorqueCal"
                           enableManualCmds := NOT "Unit1.EmNodes".unitStatus.mode.production,
                           storageCount := 30,
                           storageCycle := "Unit1.EmNodes".clock.cycle1000Msec,
                           RatedTorque := 1.27,
                           axis := "BA060AZSIDR9_SideTapeAttachmentAxisX",
                           configuration := "DriveDiagConfig".torqueLoad[9],
                           moduleInterface := "DriveDiagInterfaceHmi".torqueLoad[9]);
   "InstTorqueCal_SideTapeAttachmentAxisY"(enable := #TRUE,   // "LER_ServoTorqueCal"
                           enableManualCmds := NOT "Unit1.EmNodes".unitStatus.mode.production,
                           storageCount := 30,
                           storageCycle := "Unit1.EmNodes".clock.cycle1000Msec,
                           RatedTorque := 0.41,
                           axis := "BA060AZSIDR10_SideTapeAttachmentAxisY",
                           configuration := "DriveDiagConfig".torqueLoad[10],
                           moduleInterface := "DriveDiagInterfaceHmi".torqueLoad[10]);
END_REGION

REGION Network 7: Call: Servo Torque Cal (DR11~20)
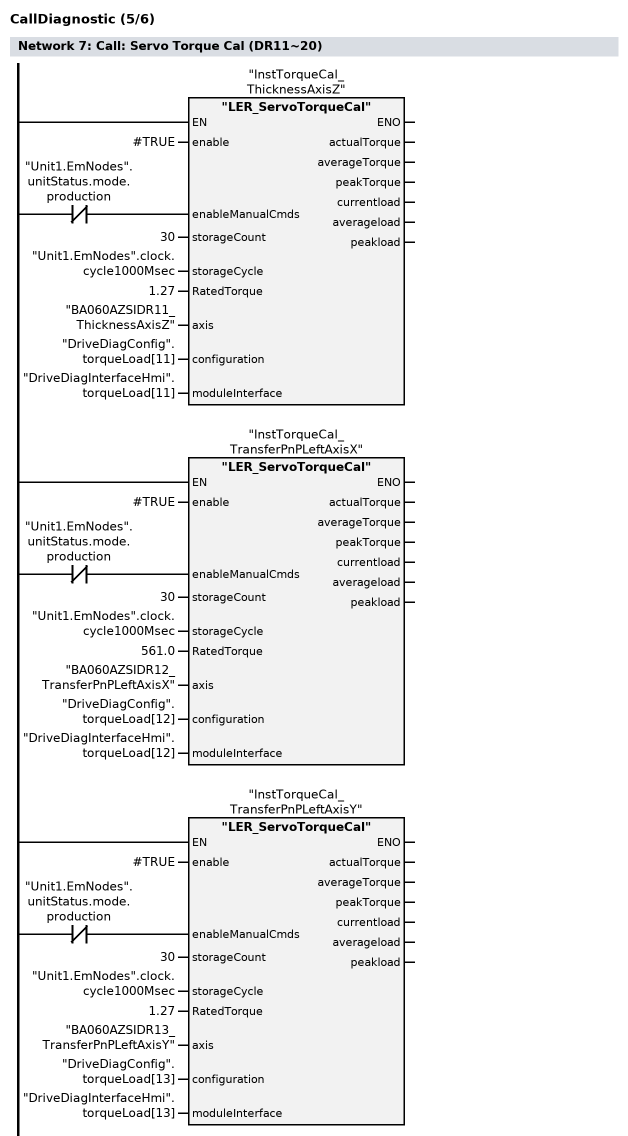
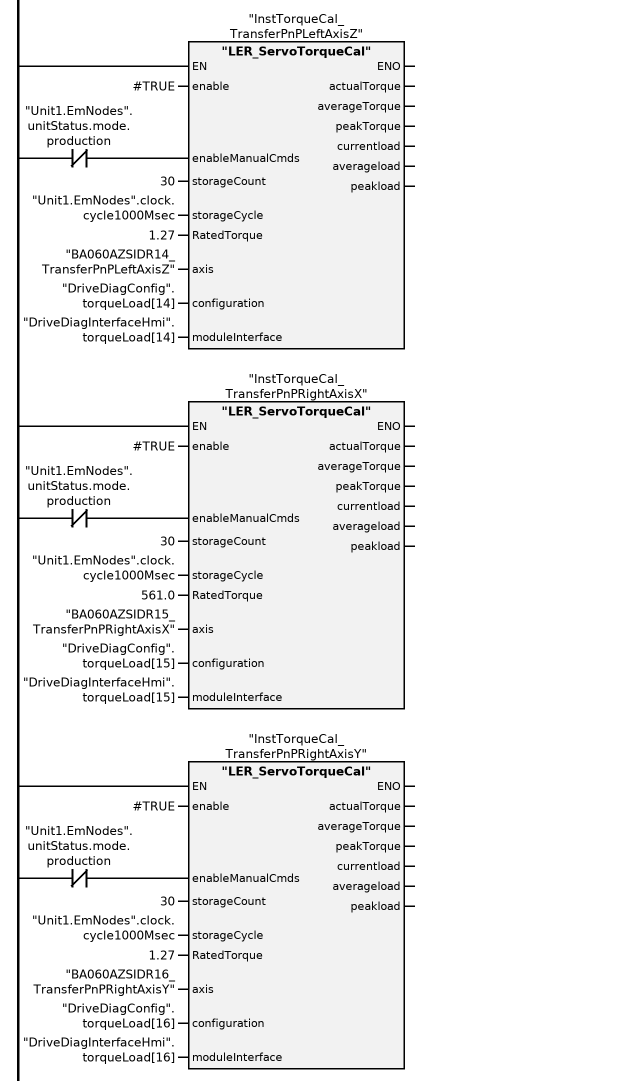
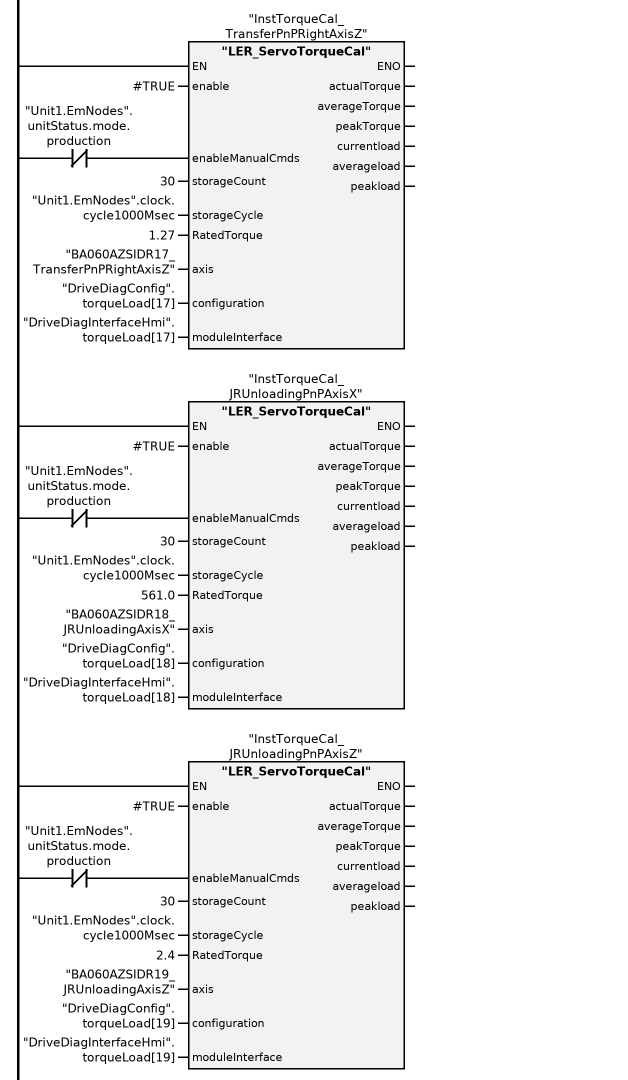
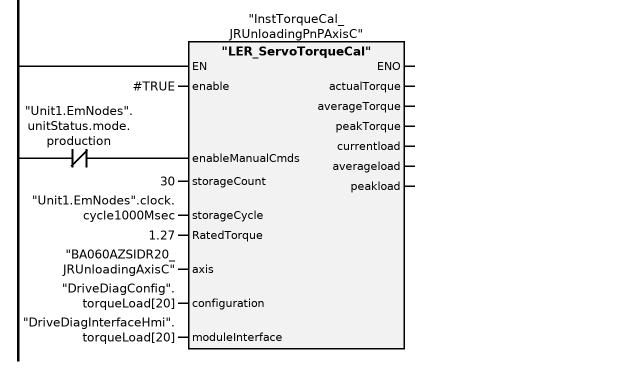
   RUNG wire#powerrail
      "InstTorqueCal_ThicknessAxisZ"(enableManualCmds := wire#w1, enable := #TRUE, storageCount := 30, storageCycle := "Unit1.EmNodes".clock.cycle1000Msec, RatedTorque := 1.27, axis := "BA060AZSIDR11_ThicknessAxisZ", configuration := "DriveDiagConfig".torqueLoad[11], moduleInterface := "DriveDiagInterfaceHmi".torqueLoad[11], actualTorque =>, averageTorque =>, peakTorque =>, currentload =>, averageload =>, peakload =>)
   END_RUNG
   RUNG wire#powerrail
      I_Contact( "Unit1.EmNodes".unitStatus.mode.production )
   END_RUNG wire#w1
   RUNG wire#powerrail
      "InstTorqueCal_TransferPnPLeftAxisX"(enableManualCmds := wire#w2, enable := #TRUE, storageCount := 30, storageCycle := "Unit1.EmNodes".clock.cycle1000Msec, RatedTorque := 561.0, axis := "BA060AZSIDR12_TransferPnPLeftAxisX", configuration := "DriveDiagConfig".torqueLoad[12], moduleInterface := "DriveDiagInterfaceHmi".torqueLoad[12], actualTorque =>, averageTorque =>, peakTorque =>, currentload =>, averageload =>, peakload =>)
   END_RUNG
   RUNG wire#powerrail
      I_Contact( "Unit1.EmNodes".unitStatus.mode.production )
   END_RUNG wire#w2
   RUNG wire#powerrail
      "InstTorqueCal_TransferPnPLeftAxisY"(enableManualCmds := wire#w3, enable := #TRUE, storageCount := 30, storageCycle := "Unit1.EmNodes".clock.cycle1000Msec, RatedTorque := 1.27, axis := "BA060AZSIDR13_TransferPnPLeftAxisY", configuration := "DriveDiagConfig".torqueLoad[13], moduleInterface := "DriveDiagInterfaceHmi".torqueLoad[13], actualTorque =>, averageTorque =>, peakTorque =>, currentload =>, averageload =>, peakload =>)
   END_RUNG
   RUNG wire#powerrail
      I_Contact( "Unit1.EmNodes".unitStatus.mode.production )
   END_RUNG wire#w3
   RUNG wire#powerrail
      "InstTorqueCal_TransferPnPLeftAxisZ"(enableManualCmds := wire#w4, enable := #TRUE, storageCount := 30, storageCycle := "Unit1.EmNodes".clock.cycle1000Msec, RatedTorque := 1.27, axis := "BA060AZSIDR14_TransferPnPLeftAxisZ", configuration := "DriveDiagConfig".torqueLoad[14], moduleInterface := "DriveDiagInterfaceHmi".torqueLoad[14], actualTorque =>, averageTorque =>, peakTorque =>, currentload =>, averageload =>, peakload =>)
   END_RUNG
   RUNG wire#powerrail
      I_Contact( "Unit1.EmNodes".unitStatus.mode.production )
   END_RUNG wire#w4
   RUNG wire#powerrail
      "InstTorqueCal_TransferPnPRightAxisX"(enableManualCmds := wire#w5, enable := #TRUE, storageCount := 30, storageCycle := "Unit1.EmNodes".clock.cycle1000Msec, RatedTorque := 561.0, axis := "BA060AZSIDR15_TransferPnPRightAxisX", configuration := "DriveDiagConfig".torqueLoad[15], moduleInterface := "DriveDiagInterfaceHmi".torqueLoad[15], actualTorque =>, averageTorque =>, peakTorque =>, currentload =>, averageload =>, peakload =>)
   END_RUNG
   RUNG wire#powerrail
      I_Contact( "Unit1.EmNodes".unitStatus.mode.production )
   END_RUNG wire#w5
   RUNG wire#powerrail
      "InstTorqueCal_TransferPnPRightAxisY"(enableManualCmds := wire#w6, enable := #TRUE, storageCount := 30, storageCycle := "Unit1.EmNodes".clock.cycle1000Msec, RatedTorque := 1.27, axis := "BA060AZSIDR16_TransferPnPRightAxisY", configuration := "DriveDiagConfig".torqueLoad[16], moduleInterface := "DriveDiagInterfaceHmi".torqueLoad[16], actualTorque =>, averageTorque =>, peakTorque =>, currentload =>, averageload =>, peakload =>)
   END_RUNG
   RUNG wire#powerrail
      I_Contact( "Unit1.EmNodes".unitStatus.mode.production )
   END_RUNG wire#w6
   RUNG wire#powerrail
      "InstTorqueCal_TransferPnPRightAxisZ"(enableManualCmds := wire#w7, enable := #TRUE, storageCount := 30, storageCycle := "Unit1.EmNodes".clock.cycle1000Msec, RatedTorque := 1.27, axis := "BA060AZSIDR17_TransferPnPRightAxisZ", configuration := "DriveDiagConfig".torqueLoad[17], moduleInterface := "DriveDiagInterfaceHmi".torqueLoad[17], actualTorque =>, averageTorque =>, peakTorque =>, currentload =>, averageload =>, peakload =>)
   END_RUNG
   RUNG wire#powerrail
      I_Contact( "Unit1.EmNodes".unitStatus.mode.production )
   END_RUNG wire#w7
   RUNG wire#powerrail
      "InstTorqueCal_JRUnloadingPnPAxisX"(enableManualCmds := wire#w8, enable := #TRUE, storageCount := 30, storageCycle := "Unit1.EmNodes".clock.cycle1000Msec, RatedTorque := 561.0, axis := "BA060AZSIDR18_JRUnloadingAxisX", configuration := "DriveDiagConfig".torqueLoad[18], moduleInterface := "DriveDiagInterfaceHmi".torqueLoad[18], actualTorque =>, averageTorque =>, peakTorque =>, currentload =>, averageload =>, peakload =>)
   END_RUNG
   RUNG wire#powerrail
      I_Contact( "Unit1.EmNodes".unitStatus.mode.production )
   END_RUNG wire#w8
   RUNG wire#powerrail
      "InstTorqueCal_JRUnloadingPnPAxisZ"(enableManualCmds := wire#w9, enable := #TRUE, storageCount := 30, storageCycle := "Unit1.EmNodes".clock.cycle1000Msec, RatedTorque := 2.4, axis := "BA060AZSIDR19_JRUnloadingAxisZ", configuration := "DriveDiagConfig".torqueLoad[19], moduleInterface := "DriveDiagInterfaceHmi".torqueLoad[19], actualTorque =>, averageTorque =>, peakTorque =>, currentload =>, averageload =>, peakload =>)
   END_RUNG
   RUNG wire#powerrail
      I_Contact( "Unit1.EmNodes".unitStatus.mode.production )
   END_RUNG wire#w9
   RUNG wire#powerrail
      "InstTorqueCal_JRUnloadingPnPAxisC"(enableManualCmds := wire#w10, enable := #TRUE, storageCount := 30, storageCycle := "Unit1.EmNodes".clock.cycle1000Msec, RatedTorque := 1.27, axis := "BA060AZSIDR20_JRUnloadingAxisC", configuration := "DriveDiagConfig".torqueLoad[20], moduleInterface := "DriveDiagInterfaceHmi".torqueLoad[20], actualTorque =>, averageTorque =>, peakTorque =>, currentload =>, averageload =>, peakload =>)
   END_RUNG
   RUNG wire#powerrail
      I_Contact( "Unit1.EmNodes".unitStatus.mode.production )
   END_RUNG wire#w10
   // the same network as SCL:
   "InstTorqueCal_ThicknessAxisZ"(enable := #TRUE,   // "LER_ServoTorqueCal"
                           enableManualCmds := NOT "Unit1.EmNodes".unitStatus.mode.production,
                           storageCount := 30,
                           storageCycle := "Unit1.EmNodes".clock.cycle1000Msec,
                           RatedTorque := 1.27,
                           axis := "BA060AZSIDR11_ThicknessAxisZ",
                           configuration := "DriveDiagConfig".torqueLoad[11],
                           moduleInterface := "DriveDiagInterfaceHmi".torqueLoad[11]);
   "InstTorqueCal_TransferPnPLeftAxisX"(enable := #TRUE,   // "LER_ServoTorqueCal"
                           enableManualCmds := NOT "Unit1.EmNodes".unitStatus.mode.production,
                           storageCount := 30,
                           storageCycle := "Unit1.EmNodes".clock.cycle1000Msec,
                           RatedTorque := 561.0,
                           axis := "BA060AZSIDR12_TransferPnPLeftAxisX",
                           configuration := "DriveDiagConfig".torqueLoad[12],
                           moduleInterface := "DriveDiagInterfaceHmi".torqueLoad[12]);
   "InstTorqueCal_TransferPnPLeftAxisY"(enable := #TRUE,   // "LER_ServoTorqueCal"
                           enableManualCmds := NOT "Unit1.EmNodes".unitStatus.mode.production,
                           storageCount := 30,
                           storageCycle := "Unit1.EmNodes".clock.cycle1000Msec,
                           RatedTorque := 1.27,
                           axis := "BA060AZSIDR13_TransferPnPLeftAxisY",
                           configuration := "DriveDiagConfig".torqueLoad[13],
                           moduleInterface := "DriveDiagInterfaceHmi".torqueLoad[13]);
   "InstTorqueCal_TransferPnPLeftAxisZ"(enable := #TRUE,   // "LER_ServoTorqueCal"
                           enableManualCmds := NOT "Unit1.EmNodes".unitStatus.mode.production,
                           storageCount := 30,
                           storageCycle := "Unit1.EmNodes".clock.cycle1000Msec,
                           RatedTorque := 1.27,
                           axis := "BA060AZSIDR14_TransferPnPLeftAxisZ",
                           configuration := "DriveDiagConfig".torqueLoad[14],
                           moduleInterface := "DriveDiagInterfaceHmi".torqueLoad[14]);
   "InstTorqueCal_TransferPnPRightAxisX"(enable := #TRUE,   // "LER_ServoTorqueCal"
                           enableManualCmds := NOT "Unit1.EmNodes".unitStatus.mode.production,
                           storageCount := 30,
                           storageCycle := "Unit1.EmNodes".clock.cycle1000Msec,
                           RatedTorque := 561.0,
                           axis := "BA060AZSIDR15_TransferPnPRightAxisX",
                           configuration := "DriveDiagConfig".torqueLoad[15],
                           moduleInterface := "DriveDiagInterfaceHmi".torqueLoad[15]);
   "InstTorqueCal_TransferPnPRightAxisY"(enable := #TRUE,   // "LER_ServoTorqueCal"
                           enableManualCmds := NOT "Unit1.EmNodes".unitStatus.mode.production,
                           storageCount := 30,
                           storageCycle := "Unit1.EmNodes".clock.cycle1000Msec,
                           RatedTorque := 1.27,
                           axis := "BA060AZSIDR16_TransferPnPRightAxisY",
                           configuration := "DriveDiagConfig".torqueLoad[16],
                           moduleInterface := "DriveDiagInterfaceHmi".torqueLoad[16]);
   "InstTorqueCal_TransferPnPRightAxisZ"(enable := #TRUE,   // "LER_ServoTorqueCal"
                           enableManualCmds := NOT "Unit1.EmNodes".unitStatus.mode.production,
                           storageCount := 30,
                           storageCycle := "Unit1.EmNodes".clock.cycle1000Msec,
                           RatedTorque := 1.27,
                           axis := "BA060AZSIDR17_TransferPnPRightAxisZ",
                           configuration := "DriveDiagConfig".torqueLoad[17],
                           moduleInterface := "DriveDiagInterfaceHmi".torqueLoad[17]);
   "InstTorqueCal_JRUnloadingPnPAxisX"(enable := #TRUE,   // "LER_ServoTorqueCal"
                           enableManualCmds := NOT "Unit1.EmNodes".unitStatus.mode.production,
                           storageCount := 30,
                           storageCycle := "Unit1.EmNodes".clock.cycle1000Msec,
                           RatedTorque := 561.0,
                           axis := "BA060AZSIDR18_JRUnloadingAxisX",
                           configuration := "DriveDiagConfig".torqueLoad[18],
                           moduleInterface := "DriveDiagInterfaceHmi".torqueLoad[18]);
   "InstTorqueCal_JRUnloadingPnPAxisZ"(enable := #TRUE,   // "LER_ServoTorqueCal"
                           enableManualCmds := NOT "Unit1.EmNodes".unitStatus.mode.production,
                           storageCount := 30,
                           storageCycle := "Unit1.EmNodes".clock.cycle1000Msec,
                           RatedTorque := 2.4,
                           axis := "BA060AZSIDR19_JRUnloadingAxisZ",
                           configuration := "DriveDiagConfig".torqueLoad[19],
                           moduleInterface := "DriveDiagInterfaceHmi".torqueLoad[19]);
   "InstTorqueCal_JRUnloadingPnPAxisC"(enable := #TRUE,   // "LER_ServoTorqueCal"
                           enableManualCmds := NOT "Unit1.EmNodes".unitStatus.mode.production,
                           storageCount := 30,
                           storageCycle := "Unit1.EmNodes".clock.cycle1000Msec,
                           RatedTorque := 1.27,
                           axis := "BA060AZSIDR20_JRUnloadingAxisC",
                           configuration := "DriveDiagConfig".torqueLoad[20],
                           moduleInterface := "DriveDiagInterfaceHmi".torqueLoad[20]);
END_REGION

REGION Network 8: Call RFID simulation
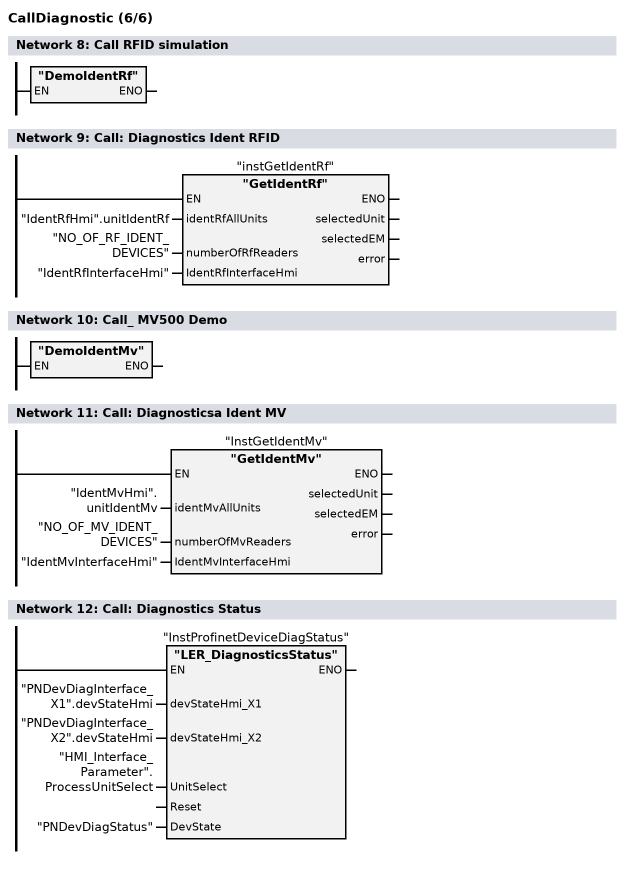
   RUNG wire#powerrail
      "DemoIdentRf"()
   END_RUNG
   // the same network as SCL:
   "DemoIdentRf"();
END_REGION

REGION Network 9: Call: Diagnostics Ident RFID
   RUNG wire#powerrail
      "instGetIdentRf"(identRfAllUnits := "IdentRfHmi".unitIdentRf, numberOfRfReaders := "NO_OF_RF_IDENT_DEVICES", IdentRfInterfaceHmi := "IdentRfInterfaceHmi", selectedUnit =>, selectedEM =>, error =>)
   END_RUNG
   // the same network as SCL:
   "instGetIdentRf"(identRfAllUnits := "IdentRfHmi".unitIdentRf,   // "GetIdentRf"
                    numberOfRfReaders := "NO_OF_RF_IDENT_DEVICES",
                    IdentRfInterfaceHmi := "IdentRfInterfaceHmi");
END_REGION

REGION Network 10: Call_ MV500 Demo
   RUNG wire#powerrail
      "DemoIdentMv"()
   END_RUNG
   // the same network as SCL:
   "DemoIdentMv"();
END_REGION

REGION Network 11: Call: Diagnosticsa Ident MV
   RUNG wire#powerrail
      "InstGetIdentMv"(identMvAllUnits := "IdentMvHmi".unitIdentMv, numberOfMvReaders := "NO_OF_MV_IDENT_DEVICES", IdentMvInterfaceHmi := "IdentMvInterfaceHmi", selectedUnit =>, selectedEM =>, error =>)
   END_RUNG
   // the same network as SCL:
   "InstGetIdentMv"(identMvAllUnits := "IdentMvHmi".unitIdentMv,   // "GetIdentMv"
                    numberOfMvReaders := "NO_OF_MV_IDENT_DEVICES",
                    IdentMvInterfaceHmi := "IdentMvInterfaceHmi");
END_REGION

REGION Network 12: Call: Diagnostics Status
   RUNG wire#powerrail
      "InstProfinetDeviceDiagStatus"(devStateHmi_X1 := "PNDevDiagInterface_X1".devStateHmi, devStateHmi_X2 := "PNDevDiagInterface_X2".devStateHmi, UnitSelect := "HMI_Interface_Parameter".ProcessUnitSelect, Reset :=, DevState := "PNDevDiagStatus")
   END_RUNG
   // the same network as SCL:
   "InstProfinetDeviceDiagStatus"(devStateHmi_X1 := "PNDevDiagInterface_X1".devStateHmi,   // "LER_DiagnosticsStatus"
                           devStateHmi_X2 := "PNDevDiagInterface_X2".devStateHmi,
                           UnitSelect := "HMI_Interface_Parameter".ProcessUnitSelect,
                           DevState := "PNDevDiagStatus");
END_REGION
END_FUNCTION

FUNCTION_BLOCK "CallInterfaceSignals"   // FB38, LAD
TITLE = CallInterfaceSignals
AUTHOR : SICAR
FAMILY : Diag
VERSION : 1.0
// The block serves as a calling interface of the block “InterfaceSignalsBool“. The block is designed as function block in order to implement the block calls as multi-instances.
// stored: IsIECCheckEnabled true, MemoryReserve 100, SetENOAutomatically true
   VAR
      statReadValueHmi : Bool;   // HMI: Read value signal
      statSelectSignalsHmi : USInt := 1;   // HMI: Selected interface signals (1..16)
      statSelectSignalsOld { ExternalAccessible := 'False'; ExternalVisible := 'False'; ExternalWritable := 'False'} : USInt;   // Old value: Selected interface signals
      statRisEdgeReadName { ExternalAccessible := 'False'; ExternalVisible := 'False'; ExternalWritable := 'False'} : Bool;   // Rising edge
      statPosPulseReadName : Bool;   // Positive pulse
      statInterfaceSignalsHmi : Array[0..100] of "typeInterfaceSignalsHmi";   // HMI: Description, value and symbolic name
      instSignals1Left { ExternalAccessible := 'False'; ExternalVisible := 'False'; ExternalWritable := 'False'} : "LAF_InterfaceSignalsBool";   // interface signals screen 1 left
      instSignals1Right { ExternalAccessible := 'False'; ExternalVisible := 'False'; ExternalWritable := 'False'} : "LAF_InterfaceSignalsBool";   // interface signals screen 1 right
      instSignals2Left { ExternalAccessible := 'False'; ExternalVisible := 'False'; ExternalWritable := 'False'} : "LAF_InterfaceSignalsBool";   // interface signals screen 2 left
      instSignals2Right { ExternalAccessible := 'False'; ExternalVisible := 'False'; ExternalWritable := 'False'} : "LAF_InterfaceSignalsBool";   // interface signals screen 2 right
      instSignals3Left { ExternalAccessible := 'False'; ExternalVisible := 'False'; ExternalWritable := 'False'} : "LAF_InterfaceSignalsBool";   // interface signals screen 3 left
      instSignals3Right { ExternalAccessible := 'False'; ExternalVisible := 'False'; ExternalWritable := 'False'} : "LAF_InterfaceSignalsBool";   // interface signals screen 3 right
      instSignals4Left { ExternalAccessible := 'False'; ExternalVisible := 'False'; ExternalWritable := 'False'} : "LAF_InterfaceSignalsBool";   // interface signals screen 4 left
      instSignals4Right { ExternalAccessible := 'False'; ExternalVisible := 'False'; ExternalWritable := 'False'} : "LAF_InterfaceSignalsBool";   // interface signals screen 4 right
      instSignals5Left { ExternalAccessible := 'False'; ExternalVisible := 'False'; ExternalWritable := 'False'} : "LAF_InterfaceSignalsBool";   // interface signals screen 5 left
      instSignals5Right { ExternalAccessible := 'False'; ExternalVisible := 'False'; ExternalWritable := 'False'} : "LAF_InterfaceSignalsBool";   // interface signals screen 5 right
      instSignals6Left { S7_SetPoint := 'True'} : "LAF_InterfaceSignalsBool";   // interface signals screen 6 left
      instSignals6Right { S7_SetPoint := 'True'} : "LAF_InterfaceSignalsBool";   // interface signals screen 6 right
      instSignals7Left { S7_SetPoint := 'True'} : "LAF_InterfaceSignalsBool";   // interface signals screen 7 left
      instSignals7Right { S7_SetPoint := 'True'} : "LAF_InterfaceSignalsBool";   // interface signals screen 7 right
      instSignals8Left { S7_SetPoint := 'True'} : "LAF_InterfaceSignalsBool";   // interface signals screen 8 left
      instSignals8Right { S7_SetPoint := 'True'} : "LAF_InterfaceSignalsBool";   // interface signals screen 8 right
      instSignals9Left { S7_SetPoint := 'True'} : "LAF_InterfaceSignalsBool";   // interface signals screen 9 left
      instSignals9Right { S7_SetPoint := 'True'} : "LAF_InterfaceSignalsBool";   // interface signals screen 9 right
      instSignals10Left_ { S7_SetPoint := 'True'} : "LAF_InterfaceSignalsBool";   // interface signals screen 10 left
      instSignals10Right { S7_SetPoint := 'True'} : "LAF_InterfaceSignalsBool";   // interface signals screen 10 right
      instSignals11Left { S7_SetPoint := 'True'} : "LAF_InterfaceSignalsBool";   // interface signals screen 11 left
      instSignals11Right { S7_SetPoint := 'True'} : "LAF_InterfaceSignalsBool";   // interface signals screen 11 right
      instSignals12Left { S7_SetPoint := 'True'} : "LAF_InterfaceSignalsBool";   // interface signals screen 12 left
      instSignals12Right { S7_SetPoint := 'True'} : "LAF_InterfaceSignalsBool";   // interface signals screen 12 right
      instSignals13Left { S7_SetPoint := 'True'} : "LAF_InterfaceSignalsBool";   // interface signals screen 13 left
      instSignals13Right { S7_SetPoint := 'True'} : "LAF_InterfaceSignalsBool";   // interface signals screen 13 right
      instSignals14Left { S7_SetPoint := 'True'} : "LAF_InterfaceSignalsBool";   // interface signals screen 14 left
      instSignals14Right { S7_SetPoint := 'True'} : "LAF_InterfaceSignalsBool";   // interface signals screen 14 right
      instSignals15Left { S7_SetPoint := 'True'} : "LAF_InterfaceSignalsBool";   // interface signals screen 15 left
      instSignals15Right { S7_SetPoint := 'True'} : "LAF_InterfaceSignalsBool";   // interface signals screen 15 right
      instSignals16Left { S7_SetPoint := 'True'} : "LAF_InterfaceSignalsBool";   // interface signals screen 16 left
      instSignals16Right { S7_SetPoint := 'True'} : "LAF_InterfaceSignalsBool";   // interface signals screen 16 right
      instSignals17Left { S7_SetPoint := 'True'} : "LAF_InterfaceSignalsBool";   // interface signals screen 17 left
      instSignals17Right { S7_SetPoint := 'True'} : "LAF_InterfaceSignalsBool";   // interface signals screen 17 right
      instSignals18Left { S7_SetPoint := 'True'} : "LAF_InterfaceSignalsBool";   // interface signals screen 18 left
      instSignals18Right { S7_SetPoint := 'True'} : "LAF_InterfaceSignalsBool";   // interface signals screen 18 right
      instSignals19Left { S7_SetPoint := 'True'} : "LAF_InterfaceSignalsBool";   // interface signals screen 19 left
      instSignals19Right { S7_SetPoint := 'True'} : "LAF_InterfaceSignalsBool";   // interface signals screen 19 right
      instSignals20Left { S7_SetPoint := 'True'} : "LAF_InterfaceSignalsBool";   // interface signals screen 20 left
      instSignals20Right { S7_SetPoint := 'True'} : "LAF_InterfaceSignalsBool";   // interface signals screen 20 right
      instSignals21Left { S7_SetPoint := 'True'} : "LAF_InterfaceSignalsBool";   // interface signals screen 21 left
      instSignals21Right { S7_SetPoint := 'True'} : "LAF_InterfaceSignalsBool";   // interface signals screen 21 right
      instSignals22Left { S7_SetPoint := 'True'} : "LAF_InterfaceSignalsBool";   // interface signals screen 22 left
      instSignals22Right { S7_SetPoint := 'True'} : "LAF_InterfaceSignalsBool";   // interface signals screen 22 right
      instSignals23Left { S7_SetPoint := 'True'} : "LAF_InterfaceSignalsBool";   // interface signals screen 23 left
      instSignals23Right { S7_SetPoint := 'True'} : "LAF_InterfaceSignalsBool";   // interface signals screen 23 right
      instSignals24Left { S7_SetPoint := 'True'} : "LAF_InterfaceSignalsBool";   // interface signals screen 24 left
      instSignals24Right { S7_SetPoint := 'True'} : "LAF_InterfaceSignalsBool";   // interface signals screen 24 right
      instSignals25Left { S7_SetPoint := 'True'} : "LAF_InterfaceSignalsBool";   // interface signals screen 25 left
      instSignals25Right { S7_SetPoint := 'True'} : "LAF_InterfaceSignalsBool";   // interface signals screen 25 right
      instSignals26Left { S7_SetPoint := 'True'} : "LAF_InterfaceSignalsBool";   // interface signals screen 26 left
      instSignals26Right { S7_SetPoint := 'True'} : "LAF_InterfaceSignalsBool";   // interface signals screen 26 right
      instSignals27Left { S7_SetPoint := 'True'} : "LAF_InterfaceSignalsBool";   // interface signals screen 27 left
      instSignals27Right { S7_SetPoint := 'True'} : "LAF_InterfaceSignalsBool";   // interface signals screen 27 right
      instSignals28Left { S7_SetPoint := 'True'} : "LAF_InterfaceSignalsBool";   // interface signals screen 28 left
      instSignals28Right { S7_SetPoint := 'True'} : "LAF_InterfaceSignalsBool";   // interface signals screen 28 right
      instSignals29Left { S7_SetPoint := 'True'} : "LAF_InterfaceSignalsBool";   // interface signals screen 29 left
      instSignals29Right { S7_SetPoint := 'True'} : "LAF_InterfaceSignalsBool";   // interface signals screen 29 right
      instSignals30Left { S7_SetPoint := 'True'} : "LAF_InterfaceSignalsBool";   // interface signals screen 30 left
      instSignals30Right { S7_SetPoint := 'True'} : "LAF_InterfaceSignalsBool";   // interface signals screen 30 right
      instSignals31Left { S7_SetPoint := 'True'} : "LAF_InterfaceSignalsBool";   // interface signals screen 31 left
      instSignals31Right { S7_SetPoint := 'True'} : "LAF_InterfaceSignalsBool";   // interface signals screen 31 right
      instSignals32Left { S7_SetPoint := 'True'} : "LAF_InterfaceSignalsBool";   // interface signals screen 32 left
      instSignals32Right { S7_SetPoint := 'True'} : "LAF_InterfaceSignalsBool";   // interface signals screen 32 right
      instSignals33Left { S7_SetPoint := 'True'} : "LAF_InterfaceSignalsBool";   // interface signals screen 33 left
      instSignals33Right { S7_SetPoint := 'True'} : "LAF_InterfaceSignalsBool";   // interface signals screen 33 right
      instSignals34Left { S7_SetPoint := 'True'} : "LAF_InterfaceSignalsBool";   // interface signals screen 34 left
      instSignals34Right { S7_SetPoint := 'True'} : "LAF_InterfaceSignalsBool";   // interface signals screen 34 right
      instSignals35Left { S7_SetPoint := 'True'} : "LAF_InterfaceSignalsBool";   // interface signals screen 35 left
      instSignals35Right { S7_SetPoint := 'True'} : "LAF_InterfaceSignalsBool";   // interface signals screen 35 right
      instSignals36Left { S7_SetPoint := 'True'} : "LAF_InterfaceSignalsBool";   // interface signals screen 36 left
      instSignals36Right { S7_SetPoint := 'True'} : "LAF_InterfaceSignalsBool";   // interface signals screen 36 right
      instSignals37Left { S7_SetPoint := 'True'} : "LAF_InterfaceSignalsBool";   // interface signals screen 37 left
      instSignals37Right { S7_SetPoint := 'True'} : "LAF_InterfaceSignalsBool";   // interface signals screen 37 right
      instSignals38Left { S7_SetPoint := 'True'} : "LAF_InterfaceSignalsBool";   // interface signals screen 38 left
      instSignals38Right { S7_SetPoint := 'True'} : "LAF_InterfaceSignalsBool";   // interface signals screen 38 right
      instSignals39Left { S7_SetPoint := 'True'} : "LAF_InterfaceSignalsBool";   // interface signals screen 39 left
      instSignals39Right { S7_SetPoint := 'True'} : "LAF_InterfaceSignalsBool";   // interface signals screen 39 right
      instSignals40Left { S7_SetPoint := 'True'} : "LAF_InterfaceSignalsBool";   // interface signals screen 40 left
      instSignals40Right { S7_SetPoint := 'True'} : "LAF_InterfaceSignalsBool";   // interface signals screen 40 right
      instSignals41Left { S7_SetPoint := 'True'} : "LAF_InterfaceSignalsBool";   // interface signals screen 41 left
      instSignals41Right { S7_SetPoint := 'True'} : "LAF_InterfaceSignalsBool";   // interface signals screen 41 right
      instSignals42Left { S7_SetPoint := 'True'} : "LAF_InterfaceSignalsBool";   // interface signals screen 42 left
      instSignals42Right { S7_SetPoint := 'True'} : "LAF_InterfaceSignalsBool";   // interface signals screen 42 right
      instSignals43Left { S7_SetPoint := 'True'} : "LAF_InterfaceSignalsBool";   // interface signals screen 43 left
      instSignals43Right { S7_SetPoint := 'True'} : "LAF_InterfaceSignalsBool";   // interface signals screen 43 right
      instSignals44Left { S7_SetPoint := 'True'} : "LAF_InterfaceSignalsBool";   // interface signals screen 44 left
      instSignals44Right { S7_SetPoint := 'True'} : "LAF_InterfaceSignalsBool";   // interface signals screen 44 right
      instSignals45Left { S7_SetPoint := 'True'} : "LAF_InterfaceSignalsBool";   // interface signals screen 45 left
      instSignals45Right { S7_SetPoint := 'True'} : "LAF_InterfaceSignalsBool";   // interface signals screen 45 right
      instSignals46Left { S7_SetPoint := 'True'} : "LAF_InterfaceSignalsBool";   // interface signals screen 46 left
      instSignals46Right { S7_SetPoint := 'True'} : "LAF_InterfaceSignalsBool";   // interface signals screen 46 right
      instSignals47Left { S7_SetPoint := 'True'} : "LAF_InterfaceSignalsBool";   // interface signals screen 47 left
      instSignals47Right { S7_SetPoint := 'True'} : "LAF_InterfaceSignalsBool";   // interface signals screen 47 right
      instSignals48Left { S7_SetPoint := 'True'} : "LAF_InterfaceSignalsBool";   // interface signals screen 48 left
      instSignals48Right { S7_SetPoint := 'True'} : "LAF_InterfaceSignalsBool";   // interface signals screen 48 right
      instSignals49Left { S7_SetPoint := 'True'} : "LAF_InterfaceSignalsBool";   // interface signals screen 49 left
      instSignals49Right { S7_SetPoint := 'True'} : "LAF_InterfaceSignalsBool";   // interface signals screen 49 right
      instSignals50Left { S7_SetPoint := 'True'} : "LAF_InterfaceSignalsBool";   // interface signals screen 50 left
      instSignals50Right { S7_SetPoint := 'True'} : "LAF_InterfaceSignalsBool";   // interface signals screen 50 right
      instSignals51Left { S7_SetPoint := 'True'} : "LAF_InterfaceSignalsBool";   // interface signals screen 51 left
      instSignals51Right { S7_SetPoint := 'True'} : "LAF_InterfaceSignalsBool";   // interface signals screen 51 right
      instSignals52Left { S7_SetPoint := 'True'} : "LAF_InterfaceSignalsBool";   // interface signals screen 52 left
      instSignals52Right { S7_SetPoint := 'True'} : "LAF_InterfaceSignalsBool";   // interface signals screen 52 right
      instSignals53Left { S7_SetPoint := 'True'} : "LAF_InterfaceSignalsBool";   // interface signals screen 53 left
      instSignals53Right { S7_SetPoint := 'True'} : "LAF_InterfaceSignalsBool";   // interface signals screen 53 right
      instSignals54Left { S7_SetPoint := 'True'} : "LAF_InterfaceSignalsBool";   // interface signals screen 54 left
      instSignals54Right { S7_SetPoint := 'True'} : "LAF_InterfaceSignalsBool";   // interface signals screen 54 right
      instSignals55Left { S7_SetPoint := 'True'} : "LAF_InterfaceSignalsBool";   // interface signals screen 55 left
      instSignals55Right { S7_SetPoint := 'True'} : "LAF_InterfaceSignalsBool";   // interface signals screen 55 right
      instSignals56Left { S7_SetPoint := 'True'} : "LAF_InterfaceSignalsBool";   // interface signals screen 56 left
      instSignals56Right { S7_SetPoint := 'True'} : "LAF_InterfaceSignalsBool";   // interface signals screen 56 right
      instSignals57Left { S7_SetPoint := 'True'} : "LAF_InterfaceSignalsBool";   // interface signals screen 57 left
      instSignals57Right { S7_SetPoint := 'True'} : "LAF_InterfaceSignalsBool";   // interface signals screen 57 right
      instSignals58Left { S7_SetPoint := 'True'} : "LAF_InterfaceSignalsBool";   // interface signals screen 58 left
      instSignals58Right { S7_SetPoint := 'True'} : "LAF_InterfaceSignalsBool";   // interface signals screen 58 right
      instSignals59Left { S7_SetPoint := 'True'} : "LAF_InterfaceSignalsBool";   // interface signals screen 59 left
      instSignals59Right { S7_SetPoint := 'True'} : "LAF_InterfaceSignalsBool";   // interface signals screen 59 right
      instSignals60Left { S7_SetPoint := 'True'} : "LAF_InterfaceSignalsBool";   // interface signals screen 60 left
      instSignals60Right { S7_SetPoint := 'True'} : "LAF_InterfaceSignalsBool";   // interface signals screen 60 right
      instSignals61Left { S7_SetPoint := 'True'} : "LAF_InterfaceSignalsBool";   // interface signals screen 61 left
      instSignals61Right { S7_SetPoint := 'True'} : "LAF_InterfaceSignalsBool";   // interface signals screen 61 right
      instSignals62Left { S7_SetPoint := 'True'} : "LAF_InterfaceSignalsBool";   // interface signals screen 62 left
      instSignals62Right { S7_SetPoint := 'True'} : "LAF_InterfaceSignalsBool";   // interface signals screen 62 right
      instSignals63Left { S7_SetPoint := 'True'} : "LAF_InterfaceSignalsBool";   // interface signals screen 63 left
      instSignals63Right { S7_SetPoint := 'True'} : "LAF_InterfaceSignalsBool";   // interface signals screen 63 right
      instSignals64Left { S7_SetPoint := 'True'} : "LAF_InterfaceSignalsBool";   // interface signals screen 64 left
      instSignals64Right { S7_SetPoint := 'True'} : "LAF_InterfaceSignalsBool";   // interface signals screen 64 right
      instSignals65Left { S7_SetPoint := 'True'} : "LAF_InterfaceSignalsBool";   // interface signals screen 65 left
      instSignals65Right { S7_SetPoint := 'True'} : "LAF_InterfaceSignalsBool";   // interface signals screen 65 right
      instSignals66Left { S7_SetPoint := 'True'} : "LAF_InterfaceSignalsBool";   // interface signals screen 66 left
      instSignals66Right { S7_SetPoint := 'True'} : "LAF_InterfaceSignalsBool";   // interface signals screen 66 right
      instSignals67Left { S7_SetPoint := 'True'} : "LAF_InterfaceSignalsBool";   // interface signals screen 67 left
      instSignals67Right { S7_SetPoint := 'True'} : "LAF_InterfaceSignalsBool";   // interface signals screen 67 right
      instSignals68Left { S7_SetPoint := 'True'} : "LAF_InterfaceSignalsBool";   // interface signals screen 68 left
      instSignals68Right { S7_SetPoint := 'True'} : "LAF_InterfaceSignalsBool";   // interface signals screen 68 right
      instSignals69Left { S7_SetPoint := 'True'} : "LAF_InterfaceSignalsBool";   // interface signals screen 69 left
      instSignals69Right { S7_SetPoint := 'True'} : "LAF_InterfaceSignalsBool";   // interface signals screen 69 right
      instSignals70Left { S7_SetPoint := 'True'} : "LAF_InterfaceSignalsBool";   // interface signals screen 70 left
      instSignals70Right { S7_SetPoint := 'True'} : "LAF_InterfaceSignalsBool";   // interface signals screen 70 right
      instSignals71Left { S7_SetPoint := 'True'} : "LAF_InterfaceSignalsBool";   // interface signals screen 71 left
      instSignals71Right { S7_SetPoint := 'True'} : "LAF_InterfaceSignalsBool";   // interface signals screen 71 right
      instSignals72Left { S7_SetPoint := 'True'} : "LAF_InterfaceSignalsBool";   // interface signals screen 72 left
      instSignals72Right { S7_SetPoint := 'True'} : "LAF_InterfaceSignalsBool";   // interface signals screen 72 right
      instSignals73Left { S7_SetPoint := 'True'} : "LAF_InterfaceSignalsBool";   // interface signals screen 73 left
      instSignals73Right { S7_SetPoint := 'True'} : "LAF_InterfaceSignalsBool";   // interface signals screen 73 right
      instSignals74Left { S7_SetPoint := 'True'} : "LAF_InterfaceSignalsBool";   // interface signals screen 74 left
      instSignals74Right { S7_SetPoint := 'True'} : "LAF_InterfaceSignalsBool";   // interface signals screen 74 right
      instSignals75Left { S7_SetPoint := 'True'} : "LAF_InterfaceSignalsBool";   // interface signals screen 75 left
      instSignals75Right { S7_SetPoint := 'True'} : "LAF_InterfaceSignalsBool";   // interface signals screen 75 right
      instSignals76Left { S7_SetPoint := 'True'} : "LAF_InterfaceSignalsBool";   // interface signals screen 76 left
      instSignals76Right { S7_SetPoint := 'True'} : "LAF_InterfaceSignalsBool";   // interface signals screen 76 right
   END_VAR
   VAR_TEMP
      tempLoopCounter : DInt;   // temp. Loop Counter
   END_VAR
   VAR_TEMP   // added for the SCL form of the ladder/FBD networks
      _w1 : Bool;
   END_VAR
BEGIN

REGION Network 1: BLOCK INFO HEADER
   // SIEMENS AG / (c)Copyright 2023
   // ------------------------------------------------------------------------------
   // Title:            CallInterfaceSignals (FB38)
   // Comment/Function: The block serves as a calling interface of the block “InterfaceSignalsBool“. The block is designed as function block in order to implement the block calls as multi-instances. 
   // Library/Family:   Diag
   // Author:           SICAR
   // Tested with:      ---
   // Engineering:      TIA Portal V19
   // Restrictions:     -
   // Requirements:     ---
   // ------------------------------------------------------------------------------
   // Change log table:
   // Version  | Date       | Expert in charge       | Changes applied
   // ---------|------------|------------------------|------------------------------
   // 01.00.00 | 11.12.2023 | SICAR
   //                         First released version
END_REGION

REGION Network 2: DESCRIPTION
   // Function block and corresponding WinCC screen are prepared for 16 data sets (“InterfaceSignals01“ through .”InterfaceSignals16“) with 32 Boolean signals each.  
   // 
   // **PLC-Data types**   
   // 
   // * LSicar_typeInterfaceSignalsBool 
   // * LSicar _typeInterfaceSignals 
   // * typeInterfaceSignalsHmi 
   // 
   // **WinCC-Faceplate**  
   // 
   // <None> 
   // 
   // **WinCC Diagnostic screen**   
   // 
   // See: ..\Library Types\LSicar_InterfaceSignalsBool.pdf  
   // 
   // **Block call example** 
   // 
   // View in ladder-logic (LAD), without parameter settings.  
   // An executable program call is available in the “SICAR-Startup” project.  
   // 
   // **Calling interface**  
   // 
   // The block is be called once in the cyclic program.  
   // 
   // **Internally used „Extended instructions / blocks“**  
   // 
   // See: ..\Library Types\LSicar_InterfaceSignalsBool.pdf
END_REGION

REGION Network 3: Initialization Loop_1
   // Preset the loop index
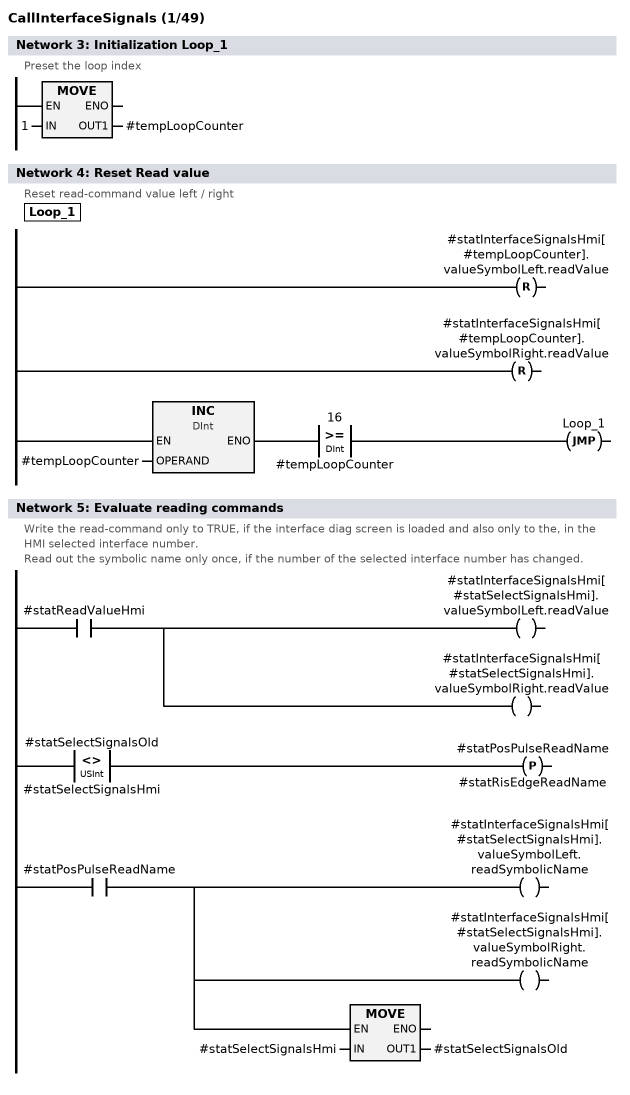
   RUNG wire#powerrail
      Move(in := 1, out1 => #tempLoopCounter)
   END_RUNG
   // the same network as SCL:
   #tempLoopCounter := 1;
END_REGION

REGION Network 4: Reset Read value
   // Reset read-command value left / right
   Label( Loop_1 )
   RUNG wire#powerrail
      R_Coil( #statInterfaceSignalsHmi[#tempLoopCounter].valueSymbolLeft.readValue )
   END_RUNG
   RUNG wire#powerrail
      R_Coil( #statInterfaceSignalsHmi[#tempLoopCounter].valueSymbolRight.readValue )
   END_RUNG
   RUNG wire#powerrail
      { S7_Templates := "DestType := DInt" } Inc( #tempLoopCounter )
      { S7_Templates := "SrcType := DInt" } GE_Contact(in1 := 16, in2 := #tempLoopCounter)
      JumpCoil( Loop_1 )
   END_RUNG
   // the same network as SCL:
   Loop_1:
   #statInterfaceSignalsHmi[#tempLoopCounter].valueSymbolLeft.readValue := FALSE;
   #statInterfaceSignalsHmi[#tempLoopCounter].valueSymbolRight.readValue := FALSE;
   #tempLoopCounter := #tempLoopCounter + 1;
   IF 16 >= #tempLoopCounter THEN GOTO Loop_1; END_IF;
END_REGION

REGION Network 5: Evaluate reading commands
   // Write the read-command only to TRUE, if the interface diag screen is loaded and also only to the, in the HMI selected interface number.
   // Read out the symbolic name only once, if the number of the selected interface number has changed.
   #statInterfaceSignalsHmi[#statSelectSignalsHmi].valueSymbolLeft.readValue := #statReadValueHmi;
   #statInterfaceSignalsHmi[#statSelectSignalsHmi].valueSymbolRight.readValue := #statReadValueHmi;
   #_w1 := #statSelectSignalsOld <> #statSelectSignalsHmi;
   #statPosPulseReadName := #_w1 AND NOT #statRisEdgeReadName;   // rising edge
   #statRisEdgeReadName := #_w1;
   #statInterfaceSignalsHmi[#statSelectSignalsHmi].valueSymbolLeft.readSymbolicName := #statPosPulseReadName;
   #statInterfaceSignalsHmi[#statSelectSignalsHmi].valueSymbolRight.readSymbolicName := #statPosPulseReadName;
   IF #statPosPulseReadName THEN #statSelectSignalsOld := #statSelectSignalsHmi; END_IF;
END_REGION

REGION Network 6: Interface Signals 01 BA030
   // Call the interface signals bool blocks of system tags
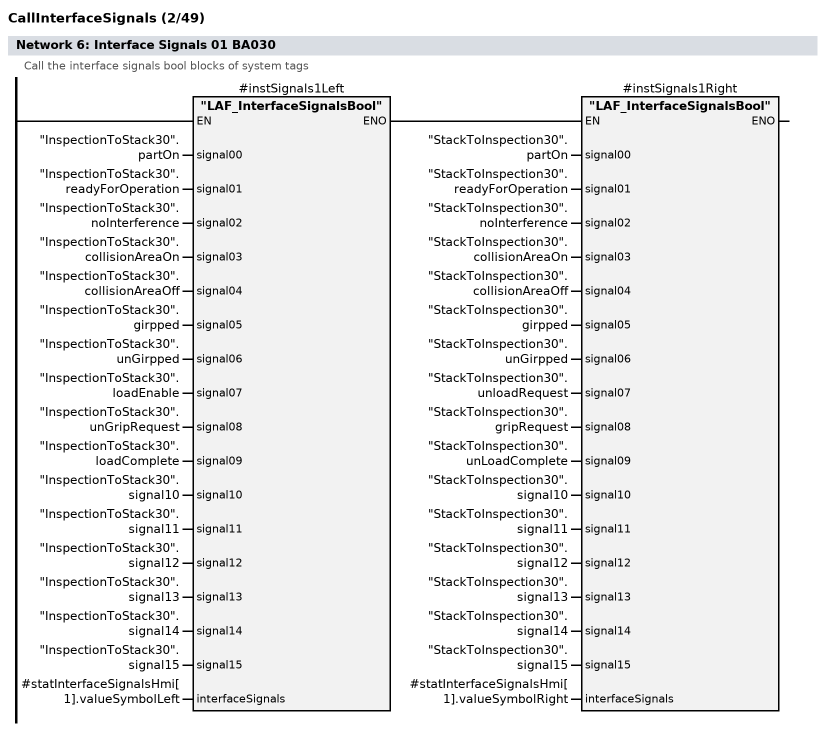
   RUNG wire#powerrail
      #instSignals1Left(signal00 := "InspectionToStack30".partOn, signal01 := "InspectionToStack30".readyForOperation, signal02 := "InspectionToStack30".noInterference, signal03 := "InspectionToStack30".collisionAreaOn, signal04 := "InspectionToStack30".collisionAreaOff, signal05 := "InspectionToStack30".girpped, signal06 := "InspectionToStack30".unGirpped, signal07 := "InspectionToStack30".loadEnable, signal08 := "InspectionToStack30".unGripRequest, signal09 := "InspectionToStack30".loadComplete, signal10 := "InspectionToStack30".signal10, signal11 := "InspectionToStack30".signal11, signal12 := "InspectionToStack30".signal12, signal13 := "InspectionToStack30".signal13, signal14 := "InspectionToStack30".signal14, signal15 := "InspectionToStack30".signal15, interfaceSignals := #statInterfaceSignalsHmi[1].valueSymbolLeft)
      #instSignals1Right(signal00 := "StackToInspection30".partOn, signal01 := "StackToInspection30".readyForOperation, signal02 := "StackToInspection30".noInterference, signal03 := "StackToInspection30".collisionAreaOn, signal04 := "StackToInspection30".collisionAreaOff, signal05 := "StackToInspection30".girpped, signal06 := "StackToInspection30".unGirpped, signal07 := "StackToInspection30".unloadRequest, signal08 := "StackToInspection30".gripRequest, signal09 := "StackToInspection30".unLoadComplete, signal10 := "StackToInspection30".signal10, signal11 := "StackToInspection30".signal11, signal12 := "StackToInspection30".signal12, signal13 := "StackToInspection30".signal13, signal14 := "StackToInspection30".signal14, signal15 := "StackToInspection30".signal15, interfaceSignals := #statInterfaceSignalsHmi[1].valueSymbolRight)
   END_RUNG
   // the same network as SCL:
   #instSignals1Left(signal00 := "InspectionToStack30".partOn,   // "LAF_InterfaceSignalsBool"
                     signal01 := "InspectionToStack30".readyForOperation,
                     signal02 := "InspectionToStack30".noInterference,
                     signal03 := "InspectionToStack30".collisionAreaOn,
                     signal04 := "InspectionToStack30".collisionAreaOff,
                     signal05 := "InspectionToStack30".girpped,
                     signal06 := "InspectionToStack30".unGirpped,
                     signal07 := "InspectionToStack30".loadEnable,
                     signal08 := "InspectionToStack30".unGripRequest,
                     signal09 := "InspectionToStack30".loadComplete,
                     signal10 := "InspectionToStack30".signal10,
                     signal11 := "InspectionToStack30".signal11,
                     signal12 := "InspectionToStack30".signal12,
                     signal13 := "InspectionToStack30".signal13,
                     signal14 := "InspectionToStack30".signal14,
                     signal15 := "InspectionToStack30".signal15,
                     interfaceSignals := #statInterfaceSignalsHmi[1].valueSymbolLeft,
                     ENO => #_w1);
   IF #_w1 THEN
       #instSignals1Right(signal00 := "StackToInspection30".partOn,   // "LAF_InterfaceSignalsBool"
                          signal01 := "StackToInspection30".readyForOperation,
                          signal02 := "StackToInspection30".noInterference,
                          signal03 := "StackToInspection30".collisionAreaOn,
                          signal04 := "StackToInspection30".collisionAreaOff,
                          signal05 := "StackToInspection30".girpped,
                          signal06 := "StackToInspection30".unGirpped,
                          signal07 := "StackToInspection30".unloadRequest,
                          signal08 := "StackToInspection30".gripRequest,
                          signal09 := "StackToInspection30".unLoadComplete,
                          signal10 := "StackToInspection30".signal10,
                          signal11 := "StackToInspection30".signal11,
                          signal12 := "StackToInspection30".signal12,
                          signal13 := "StackToInspection30".signal13,
                          signal14 := "StackToInspection30".signal14,
                          signal15 := "StackToInspection30".signal15,
                          interfaceSignals := #statInterfaceSignalsHmi[1].valueSymbolRight);
   END_IF;
END_REGION

REGION Network 7: Interface Signals 02 BA040
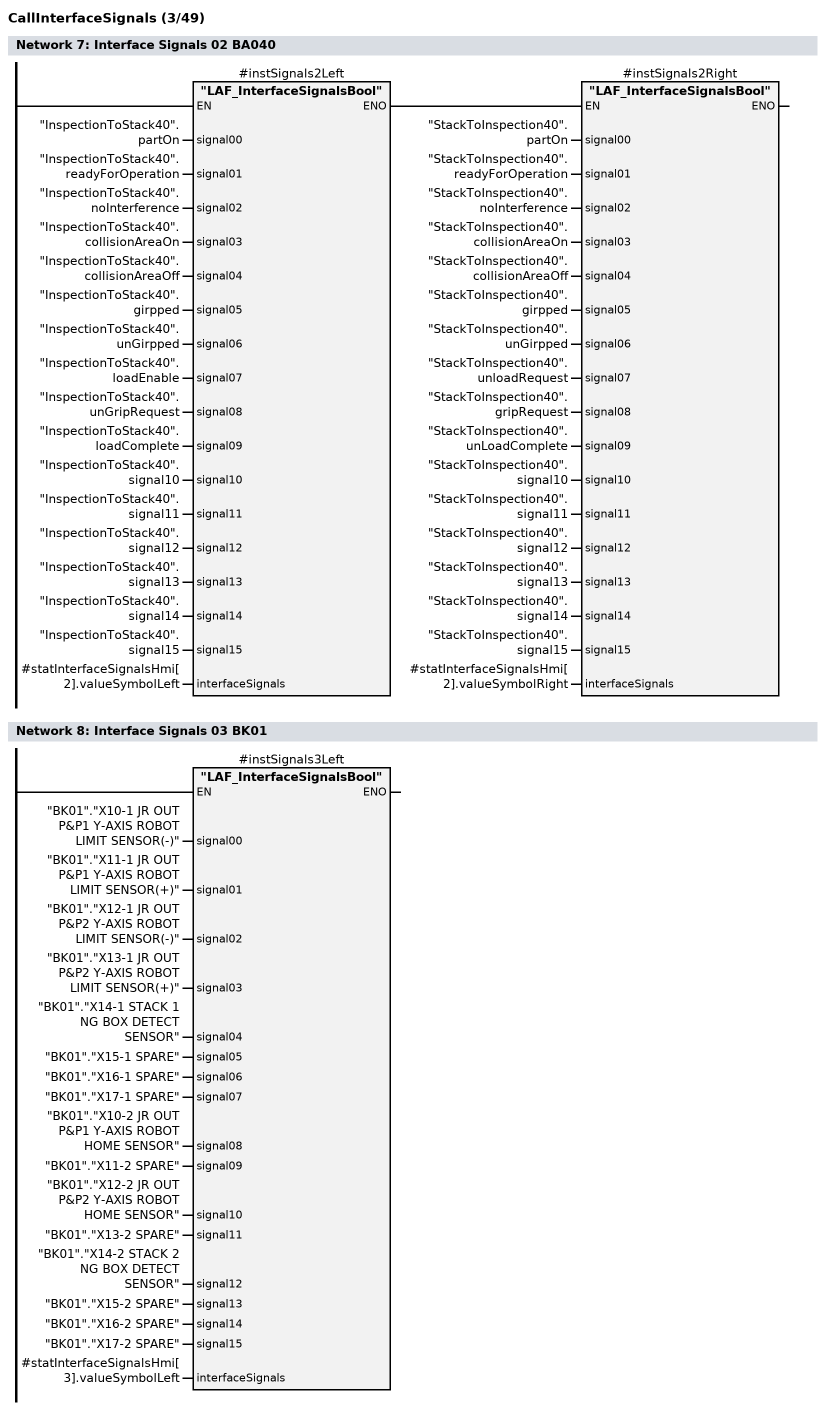
   RUNG wire#powerrail
      #instSignals2Left(signal00 := "InspectionToStack40".partOn, signal01 := "InspectionToStack40".readyForOperation, signal02 := "InspectionToStack40".noInterference, signal03 := "InspectionToStack40".collisionAreaOn, signal04 := "InspectionToStack40".collisionAreaOff, signal05 := "InspectionToStack40".girpped, signal06 := "InspectionToStack40".unGirpped, signal07 := "InspectionToStack40".loadEnable, signal08 := "InspectionToStack40".unGripRequest, signal09 := "InspectionToStack40".loadComplete, signal10 := "InspectionToStack40".signal10, signal11 := "InspectionToStack40".signal11, signal12 := "InspectionToStack40".signal12, signal13 := "InspectionToStack40".signal13, signal14 := "InspectionToStack40".signal14, signal15 := "InspectionToStack40".signal15, interfaceSignals := #statInterfaceSignalsHmi[2].valueSymbolLeft)
      #instSignals2Right(signal00 := "StackToInspection40".partOn, signal01 := "StackToInspection40".readyForOperation, signal02 := "StackToInspection40".noInterference, signal03 := "StackToInspection40".collisionAreaOn, signal04 := "StackToInspection40".collisionAreaOff, signal05 := "StackToInspection40".girpped, signal06 := "StackToInspection40".unGirpped, signal07 := "StackToInspection40".unloadRequest, signal08 := "StackToInspection40".gripRequest, signal09 := "StackToInspection40".unLoadComplete, signal10 := "StackToInspection40".signal10, signal11 := "StackToInspection40".signal11, signal12 := "StackToInspection40".signal12, signal13 := "StackToInspection40".signal13, signal14 := "StackToInspection40".signal14, signal15 := "StackToInspection40".signal15, interfaceSignals := #statInterfaceSignalsHmi[2].valueSymbolRight)
   END_RUNG
   // the same network as SCL:
   #instSignals2Left(signal00 := "InspectionToStack40".partOn,   // "LAF_InterfaceSignalsBool"
                     signal01 := "InspectionToStack40".readyForOperation,
                     signal02 := "InspectionToStack40".noInterference,
                     signal03 := "InspectionToStack40".collisionAreaOn,
                     signal04 := "InspectionToStack40".collisionAreaOff,
                     signal05 := "InspectionToStack40".girpped,
                     signal06 := "InspectionToStack40".unGirpped,
                     signal07 := "InspectionToStack40".loadEnable,
                     signal08 := "InspectionToStack40".unGripRequest,
                     signal09 := "InspectionToStack40".loadComplete,
                     signal10 := "InspectionToStack40".signal10,
                     signal11 := "InspectionToStack40".signal11,
                     signal12 := "InspectionToStack40".signal12,
                     signal13 := "InspectionToStack40".signal13,
                     signal14 := "InspectionToStack40".signal14,
                     signal15 := "InspectionToStack40".signal15,
                     interfaceSignals := #statInterfaceSignalsHmi[2].valueSymbolLeft,
                     ENO => #_w1);
   IF #_w1 THEN
       #instSignals2Right(signal00 := "StackToInspection40".partOn,   // "LAF_InterfaceSignalsBool"
                          signal01 := "StackToInspection40".readyForOperation,
                          signal02 := "StackToInspection40".noInterference,
                          signal03 := "StackToInspection40".collisionAreaOn,
                          signal04 := "StackToInspection40".collisionAreaOff,
                          signal05 := "StackToInspection40".girpped,
                          signal06 := "StackToInspection40".unGirpped,
                          signal07 := "StackToInspection40".unloadRequest,
                          signal08 := "StackToInspection40".gripRequest,
                          signal09 := "StackToInspection40".unLoadComplete,
                          signal10 := "StackToInspection40".signal10,
                          signal11 := "StackToInspection40".signal11,
                          signal12 := "StackToInspection40".signal12,
                          signal13 := "StackToInspection40".signal13,
                          signal14 := "StackToInspection40".signal14,
                          signal15 := "StackToInspection40".signal15,
                          interfaceSignals := #statInterfaceSignalsHmi[2].valueSymbolRight);
   END_IF;
END_REGION

REGION Network 8: Interface Signals 03 BK01
   RUNG wire#powerrail
      #instSignals3Left(signal00 := "BK01"."X10-1 JR OUT P&P1 Y-AXIS ROBOT LIMIT SENSOR(-)", signal01 := "BK01"."X11-1 JR OUT P&P1 Y-AXIS ROBOT LIMIT SENSOR(+)", signal02 := "BK01"."X12-1 JR OUT P&P2 Y-AXIS ROBOT LIMIT SENSOR(-)", signal03 := "BK01"."X13-1 JR OUT P&P2 Y-AXIS ROBOT LIMIT SENSOR(+)", signal04 := "BK01"."X14-1 STACK 1 NG BOX DETECT SENSOR", signal05 := "BK01"."X15-1 SPARE", signal06 := "BK01"."X16-1 SPARE", signal07 := "BK01"."X17-1 SPARE", signal08 := "BK01"."X10-2 JR OUT P&P1 Y-AXIS ROBOT HOME SENSOR", signal09 := "BK01"."X11-2 SPARE", signal10 := "BK01"."X12-2 JR OUT P&P2 Y-AXIS ROBOT HOME SENSOR", signal11 := "BK01"."X13-2 SPARE", signal12 := "BK01"."X14-2 STACK 2 NG BOX DETECT SENSOR", signal13 := "BK01"."X15-2 SPARE", signal14 := "BK01"."X16-2 SPARE", signal15 := "BK01"."X17-2 SPARE", interfaceSignals := #statInterfaceSignalsHmi[3].valueSymbolLeft)
   END_RUNG
   // the same network as SCL:
   #instSignals3Left(signal00 := "BK01"."X10-1 JR OUT P&P1 Y-AXIS ROBOT LIMIT SENSOR(-)",   // "LAF_InterfaceSignalsBool"
                     signal01 := "BK01"."X11-1 JR OUT P&P1 Y-AXIS ROBOT LIMIT SENSOR(+)",
                     signal02 := "BK01"."X12-1 JR OUT P&P2 Y-AXIS ROBOT LIMIT SENSOR(-)",
                     signal03 := "BK01"."X13-1 JR OUT P&P2 Y-AXIS ROBOT LIMIT SENSOR(+)",
                     signal04 := "BK01"."X14-1 STACK 1 NG BOX DETECT SENSOR",
                     signal05 := "BK01"."X15-1 SPARE",
                     signal06 := "BK01"."X16-1 SPARE",
                     signal07 := "BK01"."X17-1 SPARE",
                     signal08 := "BK01"."X10-2 JR OUT P&P1 Y-AXIS ROBOT HOME SENSOR",
                     signal09 := "BK01"."X11-2 SPARE",
                     signal10 := "BK01"."X12-2 JR OUT P&P2 Y-AXIS ROBOT HOME SENSOR",
                     signal11 := "BK01"."X13-2 SPARE",
                     signal12 := "BK01"."X14-2 STACK 2 NG BOX DETECT SENSOR",
                     signal13 := "BK01"."X15-2 SPARE",
                     signal14 := "BK01"."X16-2 SPARE",
                     signal15 := "BK01"."X17-2 SPARE",
                     interfaceSignals := #statInterfaceSignalsHmi[3].valueSymbolLeft);
END_REGION

REGION Network 9: Interface Signals 04 BK02
   // Call the interface signals bool blocks of opmode 4
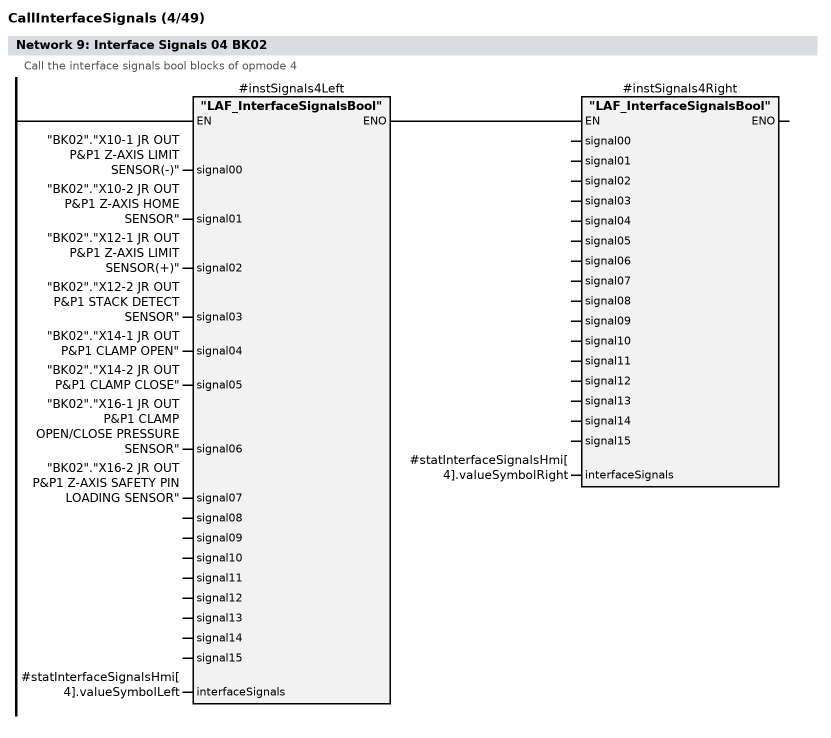
   RUNG wire#powerrail
      #instSignals4Left(signal00 := "BK02"."X10-1 JR OUT P&P1 Z-AXIS LIMIT SENSOR(-)", signal01 := "BK02"."X10-2 JR OUT P&P1 Z-AXIS HOME SENSOR", signal02 := "BK02"."X12-1 JR OUT P&P1 Z-AXIS LIMIT SENSOR(+)", signal03 := "BK02"."X12-2 JR OUT P&P1 STACK DETECT SENSOR", signal04 := "BK02"."X14-1 JR OUT P&P1 CLAMP OPEN", signal05 := "BK02"."X14-2 JR OUT P&P1 CLAMP CLOSE", signal06 := "BK02"."X16-1 JR OUT P&P1 CLAMP OPEN/CLOSE PRESSURE SENSOR", signal07 := "BK02"."X16-2 JR OUT P&P1 Z-AXIS SAFETY PIN LOADING SENSOR", signal08 :=, signal09 :=, signal10 :=, signal11 :=, signal12 :=, signal13 :=, signal14 :=, signal15 :=, interfaceSignals := #statInterfaceSignalsHmi[4].valueSymbolLeft)
      #instSignals4Right(signal00 :=, signal01 :=, signal02 :=, signal03 :=, signal04 :=, signal05 :=, signal06 :=, signal07 :=, signal08 :=, signal09 :=, signal10 :=, signal11 :=, signal12 :=, signal13 :=, signal14 :=, signal15 :=, interfaceSignals := #statInterfaceSignalsHmi[4].valueSymbolRight)
   END_RUNG
   // the same network as SCL:
   #instSignals4Left(signal00 := "BK02"."X10-1 JR OUT P&P1 Z-AXIS LIMIT SENSOR(-)",   // "LAF_InterfaceSignalsBool"
                     signal01 := "BK02"."X10-2 JR OUT P&P1 Z-AXIS HOME SENSOR",
                     signal02 := "BK02"."X12-1 JR OUT P&P1 Z-AXIS LIMIT SENSOR(+)",
                     signal03 := "BK02"."X12-2 JR OUT P&P1 STACK DETECT SENSOR",
                     signal04 := "BK02"."X14-1 JR OUT P&P1 CLAMP OPEN",
                     signal05 := "BK02"."X14-2 JR OUT P&P1 CLAMP CLOSE",
                     signal06 := "BK02"."X16-1 JR OUT P&P1 CLAMP OPEN/CLOSE PRESSURE SENSOR",
                     signal07 := "BK02"."X16-2 JR OUT P&P1 Z-AXIS SAFETY PIN LOADING SENSOR",
                     interfaceSignals := #statInterfaceSignalsHmi[4].valueSymbolLeft,
                     ENO => #_w1);
   IF #_w1 THEN
       #instSignals4Right(interfaceSignals := #statInterfaceSignalsHmi[4].valueSymbolRight);   // "LAF_InterfaceSignalsBool"
   END_IF;
END_REGION

REGION Network 10: Interface Signals 05 BK03
   // Call the interface signals bool blocks of opmode 4
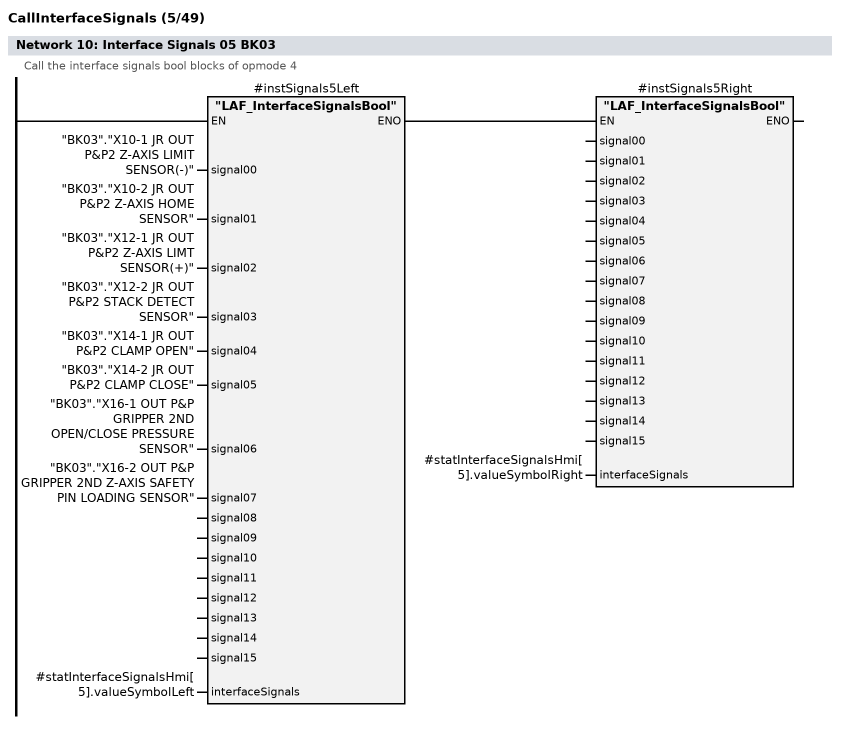
   RUNG wire#powerrail
      #instSignals5Left(signal00 := "BK03"."X10-1 JR OUT P&P2 Z-AXIS LIMIT SENSOR(-)", signal01 := "BK03"."X10-2 JR OUT P&P2 Z-AXIS HOME SENSOR", signal02 := "BK03"."X12-1 JR OUT P&P2 Z-AXIS LIMT SENSOR(+)", signal03 := "BK03"."X12-2 JR OUT P&P2 STACK DETECT SENSOR", signal04 := "BK03"."X14-1 JR OUT P&P2 CLAMP OPEN", signal05 := "BK03"."X14-2 JR OUT P&P2 CLAMP CLOSE", signal06 := "BK03"."X16-1 OUT P&P GRIPPER 2ND OPEN/CLOSE PRESSURE SENSOR", signal07 := "BK03"."X16-2 OUT P&P GRIPPER 2ND Z-AXIS SAFETY PIN LOADING SENSOR", signal08 :=, signal09 :=, signal10 :=, signal11 :=, signal12 :=, signal13 :=, signal14 :=, signal15 :=, interfaceSignals := #statInterfaceSignalsHmi[5].valueSymbolLeft)
      #instSignals5Right(signal00 :=, signal01 :=, signal02 :=, signal03 :=, signal04 :=, signal05 :=, signal06 :=, signal07 :=, signal08 :=, signal09 :=, signal10 :=, signal11 :=, signal12 :=, signal13 :=, signal14 :=, signal15 :=, interfaceSignals := #statInterfaceSignalsHmi[5].valueSymbolRight)
   END_RUNG
   // the same network as SCL:
   #instSignals5Left(signal00 := "BK03"."X10-1 JR OUT P&P2 Z-AXIS LIMIT SENSOR(-)",   // "LAF_InterfaceSignalsBool"
                     signal01 := "BK03"."X10-2 JR OUT P&P2 Z-AXIS HOME SENSOR",
                     signal02 := "BK03"."X12-1 JR OUT P&P2 Z-AXIS LIMT SENSOR(+)",
                     signal03 := "BK03"."X12-2 JR OUT P&P2 STACK DETECT SENSOR",
                     signal04 := "BK03"."X14-1 JR OUT P&P2 CLAMP OPEN",
                     signal05 := "BK03"."X14-2 JR OUT P&P2 CLAMP CLOSE",
                     signal06 := "BK03"."X16-1 OUT P&P GRIPPER 2ND OPEN/CLOSE PRESSURE SENSOR",
                     signal07 := "BK03"."X16-2 OUT P&P GRIPPER 2ND Z-AXIS SAFETY PIN LOADING SENSOR",
                     interfaceSignals := #statInterfaceSignalsHmi[5].valueSymbolLeft,
                     ENO => #_w1);
   IF #_w1 THEN
       #instSignals5Right(interfaceSignals := #statInterfaceSignalsHmi[5].valueSymbolRight);   // "LAF_InterfaceSignalsBool"
   END_IF;
END_REGION

REGION Network 11: Interface Signals 06 BK 04
   // Call the interface signals bool blocks
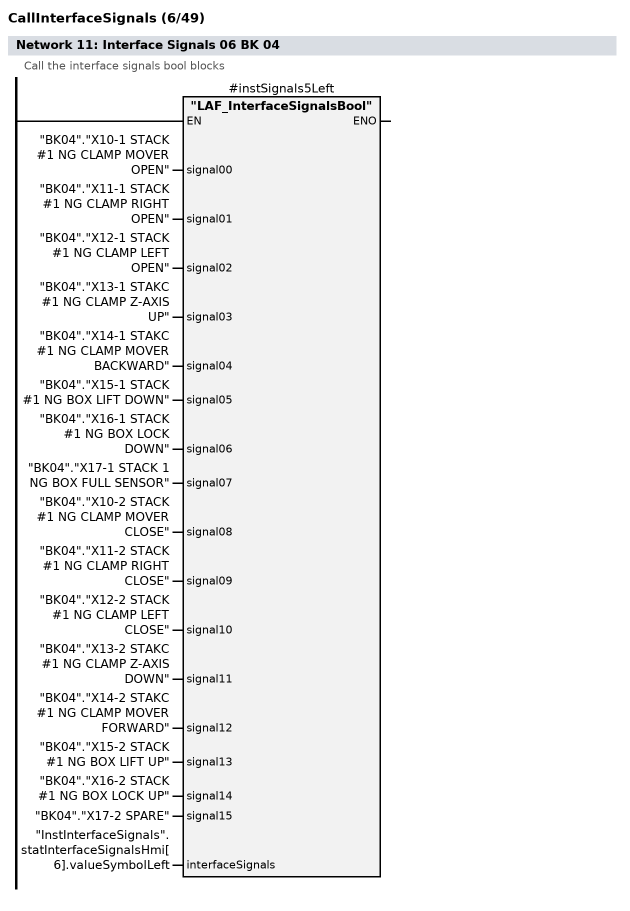
   RUNG wire#powerrail
      #instSignals5Left(signal00 := "BK04"."X10-1 STACK #1 NG CLAMP MOVER OPEN", signal01 := "BK04"."X11-1 STACK #1 NG CLAMP RIGHT OPEN", signal02 := "BK04"."X12-1 STACK #1 NG CLAMP LEFT OPEN", signal03 := "BK04"."X13-1 STAKC #1 NG CLAMP Z-AXIS UP", signal04 := "BK04"."X14-1 STAKC #1 NG CLAMP MOVER BACKWARD", signal05 := "BK04"."X15-1 STACK #1 NG BOX LIFT DOWN", signal06 := "BK04"."X16-1 STACK #1 NG BOX LOCK DOWN", signal07 := "BK04"."X17-1 STACK 1 NG BOX FULL SENSOR", signal08 := "BK04"."X10-2 STACK #1 NG CLAMP MOVER CLOSE", signal09 := "BK04"."X11-2 STACK #1 NG CLAMP RIGHT CLOSE", signal10 := "BK04"."X12-2 STACK #1 NG CLAMP LEFT CLOSE", signal11 := "BK04"."X13-2 STAKC #1 NG CLAMP Z-AXIS DOWN", signal12 := "BK04"."X14-2 STAKC #1 NG CLAMP MOVER FORWARD", signal13 := "BK04"."X15-2 STACK #1 NG BOX LIFT UP", signal14 := "BK04"."X16-2 STACK #1 NG BOX LOCK UP", signal15 := "BK04"."X17-2 SPARE", interfaceSignals := "InstInterfaceSignals".statInterfaceSignalsHmi[6].valueSymbolLeft)
   END_RUNG
   // the same network as SCL:
   #instSignals5Left(signal00 := "BK04"."X10-1 STACK #1 NG CLAMP MOVER OPEN",   // "LAF_InterfaceSignalsBool"
                     signal01 := "BK04"."X11-1 STACK #1 NG CLAMP RIGHT OPEN",
                     signal02 := "BK04"."X12-1 STACK #1 NG CLAMP LEFT OPEN",
                     signal03 := "BK04"."X13-1 STAKC #1 NG CLAMP Z-AXIS UP",
                     signal04 := "BK04"."X14-1 STAKC #1 NG CLAMP MOVER BACKWARD",
                     signal05 := "BK04"."X15-1 STACK #1 NG BOX LIFT DOWN",
                     signal06 := "BK04"."X16-1 STACK #1 NG BOX LOCK DOWN",
                     signal07 := "BK04"."X17-1 STACK 1 NG BOX FULL SENSOR",
                     signal08 := "BK04"."X10-2 STACK #1 NG CLAMP MOVER CLOSE",
                     signal09 := "BK04"."X11-2 STACK #1 NG CLAMP RIGHT CLOSE",
                     signal10 := "BK04"."X12-2 STACK #1 NG CLAMP LEFT CLOSE",
                     signal11 := "BK04"."X13-2 STAKC #1 NG CLAMP Z-AXIS DOWN",
                     signal12 := "BK04"."X14-2 STAKC #1 NG CLAMP MOVER FORWARD",
                     signal13 := "BK04"."X15-2 STACK #1 NG BOX LIFT UP",
                     signal14 := "BK04"."X16-2 STACK #1 NG BOX LOCK UP",
                     signal15 := "BK04"."X17-2 SPARE",
                     interfaceSignals := "InstInterfaceSignals".statInterfaceSignalsHmi[6].valueSymbolLeft);
END_REGION

REGION Network 12: Interface Signals 07 BK5
   // Call the interface signals bool blocks
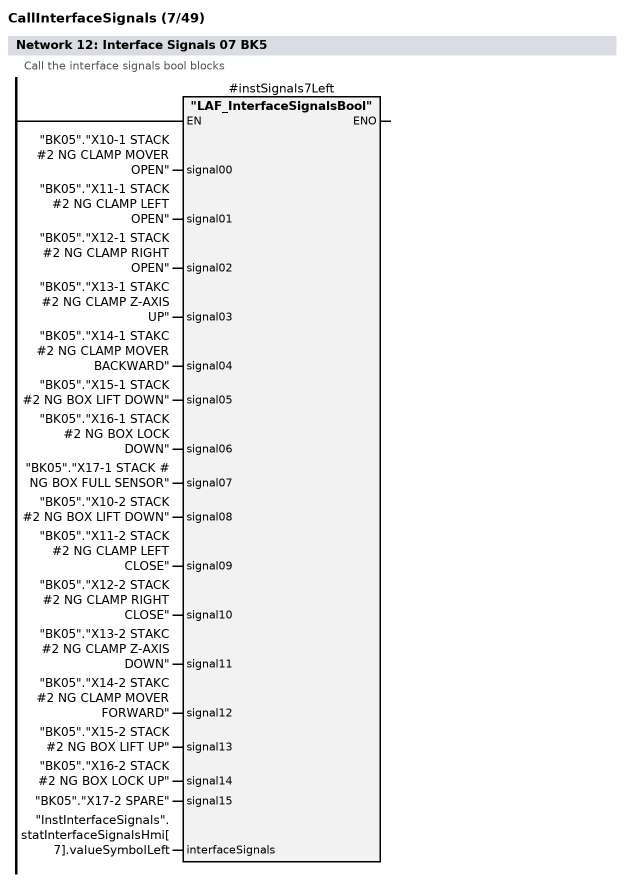
   RUNG wire#powerrail
      #instSignals7Left(signal00 := "BK05"."X10-1 STACK #2 NG CLAMP MOVER OPEN", signal01 := "BK05"."X11-1 STACK #2 NG CLAMP LEFT OPEN", signal02 := "BK05"."X12-1 STACK #2 NG CLAMP RIGHT OPEN", signal03 := "BK05"."X13-1 STAKC #2 NG CLAMP Z-AXIS UP", signal04 := "BK05"."X14-1 STAKC #2 NG CLAMP MOVER BACKWARD", signal05 := "BK05"."X15-1 STACK #2 NG BOX LIFT DOWN", signal06 := "BK05"."X16-1 STACK #2 NG BOX LOCK DOWN", signal07 := "BK05"."X17-1 STACK # NG BOX FULL SENSOR", signal08 := "BK05"."X10-2 STACK #2 NG BOX LIFT DOWN", signal09 := "BK05"."X11-2 STACK #2 NG CLAMP LEFT CLOSE", signal10 := "BK05"."X12-2 STACK #2 NG CLAMP RIGHT CLOSE", signal11 := "BK05"."X13-2 STAKC #2 NG CLAMP Z-AXIS DOWN", signal12 := "BK05"."X14-2 STAKC #2 NG CLAMP MOVER FORWARD", signal13 := "BK05"."X15-2 STACK #2 NG BOX LIFT UP", signal14 := "BK05"."X16-2 STACK #2 NG BOX LOCK UP", signal15 := "BK05"."X17-2 SPARE", interfaceSignals := "InstInterfaceSignals".statInterfaceSignalsHmi[7].valueSymbolLeft)
   END_RUNG
   // the same network as SCL:
   #instSignals7Left(signal00 := "BK05"."X10-1 STACK #2 NG CLAMP MOVER OPEN",   // "LAF_InterfaceSignalsBool"
                     signal01 := "BK05"."X11-1 STACK #2 NG CLAMP LEFT OPEN",
                     signal02 := "BK05"."X12-1 STACK #2 NG CLAMP RIGHT OPEN",
                     signal03 := "BK05"."X13-1 STAKC #2 NG CLAMP Z-AXIS UP",
                     signal04 := "BK05"."X14-1 STAKC #2 NG CLAMP MOVER BACKWARD",
                     signal05 := "BK05"."X15-1 STACK #2 NG BOX LIFT DOWN",
                     signal06 := "BK05"."X16-1 STACK #2 NG BOX LOCK DOWN",
                     signal07 := "BK05"."X17-1 STACK # NG BOX FULL SENSOR",
                     signal08 := "BK05"."X10-2 STACK #2 NG BOX LIFT DOWN",
                     signal09 := "BK05"."X11-2 STACK #2 NG CLAMP LEFT CLOSE",
                     signal10 := "BK05"."X12-2 STACK #2 NG CLAMP RIGHT CLOSE",
                     signal11 := "BK05"."X13-2 STAKC #2 NG CLAMP Z-AXIS DOWN",
                     signal12 := "BK05"."X14-2 STAKC #2 NG CLAMP MOVER FORWARD",
                     signal13 := "BK05"."X15-2 STACK #2 NG BOX LIFT UP",
                     signal14 := "BK05"."X16-2 STACK #2 NG BOX LOCK UP",
                     signal15 := "BK05"."X17-2 SPARE",
                     interfaceSignals := "InstInterfaceSignals".statInterfaceSignalsHmi[7].valueSymbolLeft);
END_REGION

REGION Network 13: Interface Signals 08 BK6
   // Call the interface signals bool blocks
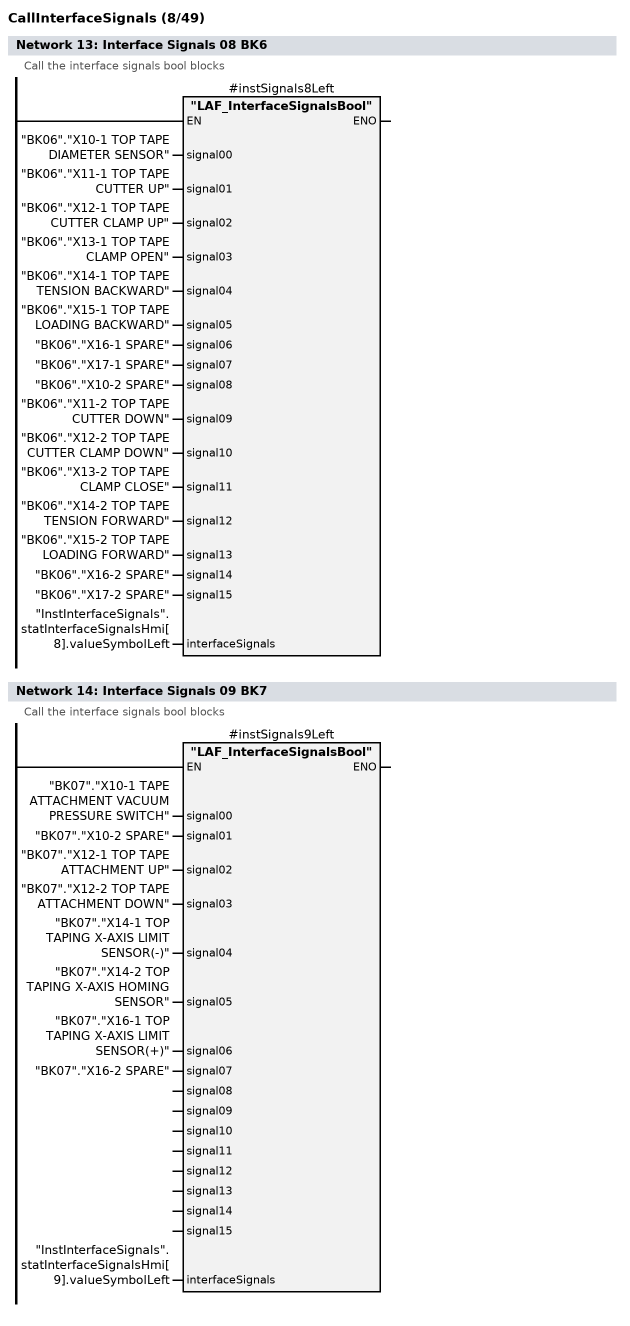
   RUNG wire#powerrail
      #instSignals8Left(signal00 := "BK06"."X10-1 TOP TAPE DIAMETER SENSOR", signal01 := "BK06"."X11-1 TOP TAPE CUTTER UP", signal02 := "BK06"."X12-1 TOP TAPE CUTTER CLAMP UP", signal03 := "BK06"."X13-1 TOP TAPE CLAMP OPEN", signal04 := "BK06"."X14-1 TOP TAPE TENSION BACKWARD", signal05 := "BK06"."X15-1 TOP TAPE LOADING BACKWARD", signal06 := "BK06"."X16-1 SPARE", signal07 := "BK06"."X17-1 SPARE", signal08 := "BK06"."X10-2 SPARE", signal09 := "BK06"."X11-2 TOP TAPE CUTTER DOWN", signal10 := "BK06"."X12-2 TOP TAPE CUTTER CLAMP DOWN", signal11 := "BK06"."X13-2 TOP TAPE CLAMP CLOSE", signal12 := "BK06"."X14-2 TOP TAPE TENSION FORWARD", signal13 := "BK06"."X15-2 TOP TAPE LOADING FORWARD", signal14 := "BK06"."X16-2 SPARE", signal15 := "BK06"."X17-2 SPARE", interfaceSignals := "InstInterfaceSignals".statInterfaceSignalsHmi[8].valueSymbolLeft)
   END_RUNG
   // the same network as SCL:
   #instSignals8Left(signal00 := "BK06"."X10-1 TOP TAPE DIAMETER SENSOR",   // "LAF_InterfaceSignalsBool"
                     signal01 := "BK06"."X11-1 TOP TAPE CUTTER UP",
                     signal02 := "BK06"."X12-1 TOP TAPE CUTTER CLAMP UP",
                     signal03 := "BK06"."X13-1 TOP TAPE CLAMP OPEN",
                     signal04 := "BK06"."X14-1 TOP TAPE TENSION BACKWARD",
                     signal05 := "BK06"."X15-1 TOP TAPE LOADING BACKWARD",
                     signal06 := "BK06"."X16-1 SPARE",
                     signal07 := "BK06"."X17-1 SPARE",
                     signal08 := "BK06"."X10-2 SPARE",
                     signal09 := "BK06"."X11-2 TOP TAPE CUTTER DOWN",
                     signal10 := "BK06"."X12-2 TOP TAPE CUTTER CLAMP DOWN",
                     signal11 := "BK06"."X13-2 TOP TAPE CLAMP CLOSE",
                     signal12 := "BK06"."X14-2 TOP TAPE TENSION FORWARD",
                     signal13 := "BK06"."X15-2 TOP TAPE LOADING FORWARD",
                     signal14 := "BK06"."X16-2 SPARE",
                     signal15 := "BK06"."X17-2 SPARE",
                     interfaceSignals := "InstInterfaceSignals".statInterfaceSignalsHmi[8].valueSymbolLeft);
END_REGION

REGION Network 14: Interface Signals 09 BK7
   // Call the interface signals bool blocks
   RUNG wire#powerrail
      #instSignals9Left(signal00 := "BK07"."X10-1 TAPE ATTACHMENT VACUUM PRESSURE SWITCH", signal01 := "BK07"."X10-2 SPARE", signal02 := "BK07"."X12-1 TOP TAPE ATTACHMENT UP", signal03 := "BK07"."X12-2 TOP TAPE ATTACHMENT DOWN", signal04 := "BK07"."X14-1 TOP TAPING X-AXIS LIMIT SENSOR(-)", signal05 := "BK07"."X14-2 TOP TAPING X-AXIS HOMING SENSOR", signal06 := "BK07"."X16-1 TOP TAPING X-AXIS LIMIT SENSOR(+)", signal07 := "BK07"."X16-2 SPARE", signal08 :=, signal09 :=, signal10 :=, signal11 :=, signal12 :=, signal13 :=, signal14 :=, signal15 :=, interfaceSignals := "InstInterfaceSignals".statInterfaceSignalsHmi[9].valueSymbolLeft)
   END_RUNG
   // the same network as SCL:
   #instSignals9Left(signal00 := "BK07"."X10-1 TAPE ATTACHMENT VACUUM PRESSURE SWITCH",   // "LAF_InterfaceSignalsBool"
                     signal01 := "BK07"."X10-2 SPARE",
                     signal02 := "BK07"."X12-1 TOP TAPE ATTACHMENT UP",
                     signal03 := "BK07"."X12-2 TOP TAPE ATTACHMENT DOWN",
                     signal04 := "BK07"."X14-1 TOP TAPING X-AXIS LIMIT SENSOR(-)",
                     signal05 := "BK07"."X14-2 TOP TAPING X-AXIS HOMING SENSOR",
                     signal06 := "BK07"."X16-1 TOP TAPING X-AXIS LIMIT SENSOR(+)",
                     signal07 := "BK07"."X16-2 SPARE",
                     interfaceSignals := "InstInterfaceSignals".statInterfaceSignalsHmi[9].valueSymbolLeft);
END_REGION

